KUKA KRL program: MyProgram_315().src

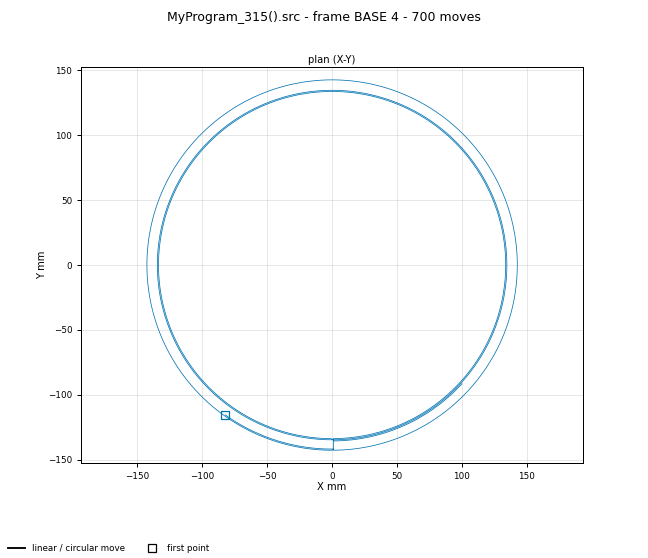
[picture p0: tool path of MyProgram_315().src in frame BASE 4, 700 of 700 moves have a stored position in this frame; points joined in program order, loops and branches not executed]
&ACCESS RVP
&REL 1
&PARAM TEMPLATE = C:\KRC\Roboter\Template\vorgabe
&PARAM EDITMASK = *
DEF MyProgram_315()
; ---- Setting reference (Base) ----
$BASE = BASE_DATA[4]

; --------------------------
; ---- Setting tool (TCP) ----
$TOOL = TOOL_DATA[3]
; --------------------------

$VEL.CP = VEL_APROX_PRINT
Startdeposition()
$VEL.CP = VEL_PRINT
LIN {X -82.35,Y -115.3687,Z 183,A -120.2522,B 3.9379,C 0.3327,E1 3.862,E2 213.1284} C_DIS
LIN {X -78.6424,Y -117.9272,Z 183,A -118.3809,B 3.9377,C 0.335,E1 3.8664,E2 211.2503} C_DIS
LIN {X -74.8735,Y -120.3553,Z 183,A -116.5285,B 3.9375,C 0.3372,E1 3.8708,E2 209.3924} C_DIS
LIN {X -70.8124,Y -122.7888,Z 183,A -114.6076,B 3.9373,C 0.3397,E1 3.8754,E2 207.4704} C_DIS
LIN {X -66.6703,Y -125.0867,Z 183,A -112.6373,B 3.9372,C 0.3416,E1 3.8802,E2 205.4924} C_DIS
LIN {X -63.0372,Y -126.954,Z 183,A -111.0289,B 3.937,C 0.3439,E1 3.8842,E2 203.8895} C_DIS
LIN {X -59.8265,Y -128.4982,Z 183,A -109.6089,B 3.9368,C 0.3456,E1 3.8878,E2 202.4722} C_DIS
LIN {X -56.4905,Y -129.9991,Z 183,A -108.1124,B 3.9367,C 0.3469,E1 3.8917,E2 200.973} C_DIS
LIN {X -53.5251,Y -131.2489,Z 183,A -106.7255,B 3.9367,C 0.3475,E1 3.8953,E2 199.5741} C_DIS
LIN {X -50.6002,Y -132.4053,Z 183,A -105.0533,B 3.9368,C 0.3452,E1 3.8998,E2 197.8465} C_DIS
LIN {X -46.7841,Y -133.7994,Z 183,A -103.1176,B 3.937,C 0.344,E1 3.905,E2 195.8696} C_DIS
LIN {X -41.3585,Y -135.5743,Z 183,A -101.5599,B 3.9362,C 0.3521,E1 3.9089,E2 194.4151} C_DIS
LIN {X -37.5342,Y -136.6841,Z 183,A -99.8325,B 3.9362,C 0.3521,E1 3.9136,E2 192.6712} C_DIS
LIN {X -34.185,Y -137.5602,Z 183,A -98.3691,B 3.9362,C 0.3523,E1 3.9176,E2 191.1985} C_DIS
LIN {X -30.1731,Y -138.494,Z 183,A -96.764,B 3.9362,C 0.3537,E1 3.9219,E2 189.6012} C_DIS
LIN {X -27.0139,Y -139.1451,Z 183,A -95.4028,B 3.9361,C 0.3537,E1 3.9257,E2 188.2317} C_DIS
LIN {X -23.267,Y -139.8199,Z 183,A -93.8958,B 3.9361,C 0.3545,E1 3.9298,E2 186.7286} C_DIS
LIN {X -18.7889,Y -140.4923,Z 183,A -92.1155,B 3.9359,C 0.3554,E1 3.9347,E2 184.9545} C_DIS
LIN {X -15.1936,Y -140.926,Z 183,A -90.5618,B 3.9359,C 0.3548,E1 3.9391,E2 183.3878} C_DIS
LIN {X -10.7309,Y -141.3366,Z 183,A -88.786,B 3.9359,C 0.3553,E1 3.944,E2 181.6162} C_DIS
LIN {X -6.3939,Y -141.6004,Z 183,A -86.9641,B 3.936,C 0.3547,E1 3.9491,E2 179.7846} C_DIS
LIN {X -2.1357,Y -141.7269,Z 183,A -85.3236,B 3.936,C 0.3554,E1 3.9537,E2 178.1545} C_DIS
LIN {X 0.9913,Y -141.7363,Z 183,A -84.3134,B 3.9357,C 0.3576,E1 3.9564,E2 177.1786} C_DIS
Enddeposition()
LIN {X 0.9913,Y -141.7363,Z 183,A -84.3134,B 3.9357,C 0.3576,E1 3.9564,E2 177.1786} C_DIS
Startdeposition()
$VEL.CP = VEL_PRINT
LIN {X 0.0025,Y -142.646,Z 183,A -85.0932,B 3.9352,C 0.3635,E1 3.954,E2 178.0429} C_DIS
LIN {X -3.4938,Y -142.6018,Z 183,A -86.4866,B 3.9352,C 0.3635,E1 3.9501,E2 179.4354} C_DIS
LIN {X -7.7044,Y -142.4366,Z 183,A -88.2171,B 3.9352,C 0.3639,E1 3.9453,E2 181.1718} C_DIS
LIN {X -11.5276,Y -142.178,Z 183,A -89.6214,B 3.9353,C 0.3626,E1 3.9414,E2 182.5582} C_DIS
LIN {X -15.0099,Y -141.852,Z 183,A -91.2226,B 3.9352,C 0.3642,E1 3.9369,E2 184.1869} C_DIS
LIN {X -19.1891,Y -141.3486,Z 183,A -92.7975,B 3.9352,C 0.3628,E1 3.9325,E2 185.7466} C_DIS
LIN {X -22.6498,Y -140.8363,Z 183,A -94.2297,B 3.9353,C 0.3626,E1 3.9286,E2 187.183} C_DIS
LIN {X -26.1124,Y -140.2348,Z 183,A -95.5706,B 3.9354,C 0.3615,E1 3.9249,E2 188.5147} C_DIS
LIN {X -28.8416,Y -139.698,Z 183,A -96.7574,B 3.9354,C 0.3616,E1 3.9216,E2 189.7113} C_DIS
LIN {X -32.9469,Y -138.7873,Z 183,A -98.6018,B 3.9354,C 0.3622,E1 3.9166,E2 191.5776} C_DIS
LIN {X -37.3426,Y -137.6701,Z 183,A -100.2942,B 3.9355,C 0.36,E1 3.912,E2 193.2527} C_DIS
LIN {X -40.2563,Y -136.8452,Z 183,A -101.5751,B 3.9355,C 0.3597,E1 3.9086,E2 194.5428} C_DIS
LIN {X -44.0427,Y -135.6755,Z 183,A -103.2725,B 3.9355,C 0.3595,E1 3.904,E2 196.2551} C_DIS
LIN {X -47.9851,Y -134.3307,Z 183,A -104.957,B 3.9357,C 0.3583,E1 3.8996,E2 197.9415} C_DIS
LIN {X -52.2995,Y -132.7114,Z 183,A -106.8391,B 3.9358,C 0.3569,E1 3.8946,E2 199.8282} C_DIS
LIN {X -56.8493,Y -130.8256,Z 183,A -108.7188,B 3.9361,C 0.3541,E1 3.8898,E2 201.6946} C_DIS
LIN {X -60.1958,Y -129.3202,Z 183,A -110.1929,B 3.9362,C 0.3526,E1 3.8861,E2 203.1689} C_DIS
LIN {X -63.3431,Y -127.8078,Z 183,A -111.6692,B 3.9362,C 0.3516,E1 3.8823,E2 204.6555} C_DIS
LIN {X -66.7705,Y -126.0518,Z 183,A -113.1503,B 3.9365,C 0.3493,E1 3.8787,E2 206.1278} C_DIS
LIN {X -70.1777,Y -124.1889,Z 183,A -114.8685,B 3.9365,C 0.3486,E1 3.8744,E2 207.8677} C_DIS
LIN {X -74.0833,Y -121.8994,Z 183,A -116.7206,B 3.9368,C 0.3464,E1 3.87,E2 209.7245} C_DIS
LIN {X -77.9926,Y -119.4361,Z 183,A -118.634,B 3.937,C 0.3442,E1 3.8655,E2 211.6458} C_DIS
LIN {X -81.8387,Y -116.8345,Z 183,A -120.4887,B 3.9372,C 0.3413,E1 3.8612,E2 213.499} C_DIS
LIN {X -85.3766,Y -114.2741,Z 183,A -122.2549,B 3.9374,C 0.3387,E1 3.8572,E2 215.2667} C_DIS
LIN {X -88.7267,Y -111.6928,Z 183,A -124.0258,B 3.9376,C 0.3364,E1 3.8533,E2 217.0474} C_DIS
LIN {X -92.1116,Y -108.9187,Z 183,A -125.838,B 3.9378,C 0.3338,E1 3.8494,E2 218.8669} C_DIS
LIN {X -95.4102,Y -106.041,Z 183,A -127.6362,B 3.9381,C 0.331,E1 3.8456,E2 220.6702} C_DIS
LIN {X -98.7395,Y -102.9478,Z 183,A -129.4764,B 3.9384,C 0.3277,E1 3.8419,E2 222.5122} C_DIS
LIN {X -101.9675,Y -99.7514,Z 183,A -131.3683,B 3.9386,C 0.3247,E1 3.8381,E2 224.4129} C_DIS
LIN {X -105.0998,Y -96.4454,Z 183,A -133.2356,B 3.9389,C 0.3213,E1 3.8346,E2 226.285} C_DIS
LIN {X -108.0049,Y -93.1807,Z 183,A -135.0551,B 3.9391,C 0.3181,E1 3.8312,E2 228.1127} C_DIS
LIN {X -111.047,Y -89.5335,Z 183,A -136.9938,B 3.9394,C 0.3143,E1 3.8278,E2 230.0551} C_DIS
LIN {X -113.7384,Y -86.0888,Z 183,A -138.7532,B 3.9397,C 0.3105,E1 3.8248,E2 231.8145} C_DIS
LIN {X -116.1196,Y -82.8489,Z 183,A -140.472,B 3.94,C 0.3076,E1 3.8219,E2 233.5468} C_DIS
LIN {X -118.6043,Y -79.2509,Z 183,A -142.2794,B 3.9403,C 0.304,E1 3.8191,E2 235.3604} C_DIS
LIN {X -120.9833,Y -75.5697,Z 183,A -144.079,B 3.9406,C 0.3001,E1 3.8164,E2 237.1648} C_DIS
LIN {X -123.2396,Y -71.8322,Z 183,A -145.927,B 3.9408,C 0.2965,E1 3.8137,E2 239.0248} C_DIS
LIN {X -125.38,Y -68.0268,Z 183,A -147.754,B 3.9411,C 0.2928,E1 3.8112,E2 240.8609} C_DIS
LIN {X -127.2528,Y -64.4509,Z 183,A -149.3448,B 3.9414,C 0.2885,E1 3.8092,E2 242.4468} C_DIS
LIN {X -128.9483,Y -60.9897,Z 183,A -150.9313,B 3.9417,C 0.2849,E1 3.8073,E2 244.0378} C_DIS
LIN {X -130.8258,Y -56.849,Z 183,A -152.914,B 3.9419,C 0.2812,E1 3.805,E2 246.0406} C_DIS
LIN {X -132.709,Y -52.3057,Z 183,A -154.9212,B 3.9423,C 0.2763,E1 3.8029,E2 248.0512} C_DIS
LIN {X -134.059,Y -48.7388,Z 183,A -156.5536,B 3.9425,C 0.2729,E1 3.8013,E2 249.6962} C_DIS
LIN {X -135.6246,Y -44.2019,Z 183,A -158.4657,B 3.9429,C 0.2677,E1 3.7996,E2 251.6052} C_DIS
LIN {X -136.7083,Y -40.7239,Z 183,A -159.9347,B 3.9431,C 0.2638,E1 3.7984,E2 253.0743} C_DIS
LIN {X -137.6658,Y -37.3588,Z 183,A -161.4756,B 3.9433,C 0.2608,E1 3.7973,E2 254.6323} C_DIS
LIN {X -138.7197,Y -33.2272,Z 183,A -163.1937,B 3.9436,C 0.2562,E1 3.7961,E2 256.3502} C_DIS
LIN {X -139.5524,Y -29.5406,Z 183,A -164.7326,B 3.9439,C 0.2521,E1 3.7952,E2 257.8909} C_DIS
LIN {X -140.2412,Y -26.079,Z 183,A -166.1968,B 3.9441,C 0.2485,E1 3.7944,E2 259.3605} C_DIS
LIN {X -140.8371,Y -22.6452,Z 183,A -167.6697,B 3.9444,C 0.2451,E1 3.7937,E2 260.8422} C_DIS
LIN {X -141.3475,Y -19.1975,Z 183,A -169.1215,B 3.9446,C 0.2415,E1 3.7931,E2 262.3001} C_DIS
LIN {X -141.7733,Y -15.7415,Z 183,A -170.5705,B 3.9448,C 0.2378,E1 3.7927,E2 263.7548} C_DIS
LIN {X -142.1148,Y -12.2755,Z 183,A -172.1312,B 3.945,C 0.2349,E1 3.7923,E2 265.3359} C_DIS
LIN {X -142.4358,Y -7.7214,Z 183,A -173.9354,B 3.9453,C 0.2295,E1 3.792,E2 267.135} C_DIS
LIN {X -142.5818,Y -4.2146,Z 183,A -175.3855,B 3.9455,C 0.2258,E1 3.7918,E2 268.5895} C_DIS
LIN {X -142.6476,Y -0.0075,Z 183,A -177.2034,B 3.9457,C 0.2218,E1 3.7918,E2 270.4232} C_DIS
LIN {X -142.6022,Y 3.4816,Z 183,A -178.6021,B 3.946,C 0.2178,E1 3.7918,E2 271.8204} C_DIS
LIN {X -142.441,Y 7.6183,Z 183,A 179.6198,B 3.9462,C 0.2138,E1 3.7921,E2 273.6124} C_DIS
LIN {X -142.1829,Y 11.4694,Z 183,A 178.1477,B 3.9464,C 0.2089,E1 3.7924,E2 275.0731} C_DIS
LIN {X -141.853,Y 15.0013,Z 183,A 176.5928,B 3.9466,C 0.2057,E1 3.7928,E2 276.644} C_DIS
LIN {X -141.3507,Y 19.1732,Z 183,A 174.8586,B 3.9468,C 0.2012,E1 3.7934,E2 278.3831} C_DIS
LIN {X -140.839,Y 22.6328,Z 183,A 173.4049,B 3.947,C 0.1976,E1 3.794,E2 279.8421} C_DIS
LIN {X -140.2388,Y 26.0914,Z 183,A 171.9887,B 3.9472,C 0.1937,E1 3.7947,E2 281.258} C_DIS
LIN {X -139.7058,Y 28.8029,Z 183,A 170.6646,B 3.9472,C 0.1919,E1 3.7955,E2 282.6092} C_DIS
LIN {X -138.7838,Y 32.9616,Z 183,A 168.8567,B 3.9475,C 0.1877,E1 3.7966,E2 284.4284} C_DIS
LIN {X -137.6667,Y 37.3555,Z 183,A 167.1157,B 3.9477,C 0.1823,E1 3.7978,E2 286.1576} C_DIS
LIN {X -136.7077,Y 40.7259,Z 183,A 165.6559,B 3.9479,C 0.1788,E1 3.799,E2 287.6231} C_DIS
LIN {X -135.6654,Y 44.0741,Z 183,A 164.0332,B 3.948,C 0.1762,E1 3.8004,E2 289.2725} C_DIS
LIN {X -134.3034,Y 48.061,Z 183,A 162.3117,B 3.9482,C 0.1719,E1 3.802,E2 290.9964} C_DIS
LIN {X -132.7108,Y 52.3011,Z 183,A 160.4077,B 3.9484,C 0.1676,E1 3.8039,E2 292.9099} C_DIS
LIN {X -130.8262,Y 56.848,Z 183,A 158.4915,B 3.9486,C 0.1621,E1 3.806,E2 294.8166} C_DIS
LIN {X -129.3279,Y 60.1791,Z 183,A 156.9927,B 3.9488,C 0.1585,E1 3.8077,E2 296.3183} C_DIS
LIN {X -127.8035,Y 63.3516,Z 183,A 155.477,B 3.9488,C 0.1556,E1 3.8096,E2 297.846} C_DIS
LIN {X -126.0351,Y 66.8022,Z 183,A 153.8636,B 3.949,C 0.152,E1 3.8117,E2 299.4654} C_DIS
LIN {X -123.933,Y 70.6278,Z 183,A 152.0311,B 3.9492,C 0.1482,E1 3.8142,E2 301.3067} C_DIS
LIN {X -121.6294,Y 74.525,Z 183,A 150.1752,B 3.9493,C 0.1441,E1 3.8169,E2 303.166} C_DIS
LIN {X -119.2914,Y 78.2133,Z 183,A 148.3566,B 3.9495,C 0.1403,E1 3.8196,E2 304.9915} C_DIS
LIN {X -116.8404,Y 81.8303,Z 183,A 146.541,B 3.9495,C 0.1367,E1 3.8225,E2 306.8134} C_DIS
LIN {X -114.2644,Y 85.3897,Z 183,A 144.7443,B 3.9497,C 0.1329,E1 3.8255,E2 308.6128} C_DIS
LIN {X -111.6942,Y 88.7248,Z 183,A 142.9703,B 3.9498,C 0.1297,E1 3.8285,E2 310.3959} C_DIS
LIN {X -108.9229,Y 92.1066,Z 183,A 141.1455,B 3.9499,C 0.1263,E1 3.8318,E2 312.2281} C_DIS
LIN {X -106.0397,Y 95.4115,Z 183,A 139.3422,B 3.95,C 0.1229,E1 3.8352,E2 314.0353} C_DIS
LIN {X -102.9541,Y 98.7329,Z 183,A 137.5179,B 3.9502,C 0.1193,E1 3.8387,E2 315.8587} C_DIS
LIN {X -99.8794,Y 101.8419,Z 183,A 135.7103,B 3.9502,C 0.1162,E1 3.8422,E2 317.6714} C_DIS
LIN {X -96.7026,Y 104.8634,Z 183,A 133.8965,B 3.9503,C 0.1132,E1 3.846,E2 319.4905} C_DIS
LIN {X -93.443,Y 107.7789,Z 183,A 132.023,B 3.9503,C 0.1108,E1 3.8499,E2 321.3775} C_DIS
LIN {X -89.8188,Y 110.8168,Z 183,A 130.146,B 3.9505,C 0.1073,E1 3.8539,E2 323.2502} C_DIS
LIN {X -86.3706,Y 113.525,Z 183,A 128.3193,B 3.9505,C 0.1048,E1 3.858,E2 325.0839} C_DIS
LIN {X -82.8502,Y 116.1186,Z 183,A 126.5424,B 3.9506,C 0.1021,E1 3.862,E2 326.8622} C_DIS
LIN {X -79.2527,Y 118.6031,Z 183,A 124.7541,B 3.9506,C 0.0996,E1 3.8662,E2 328.6532} C_DIS
LIN {X -75.5677,Y 120.9846,Z 183,A 122.9716,B 3.9508,C 0.0972,E1 3.8704,E2 330.437} C_DIS
LIN {X -71.8261,Y 123.2431,Z 183,A 121.146,B 3.9508,C 0.0953,E1 3.8748,E2 332.2703} C_DIS
LIN {X -68.0166,Y 125.3855,Z 183,A 119.3457,B 3.9508,C 0.0933,E1 3.8792,E2 334.075} C_DIS
LIN {X -64.4622,Y 127.247,Z 183,A 117.7885,B 3.9509,C 0.0909,E1 3.883,E2 335.624} C_DIS
LIN {X -60.9768,Y 128.9545,Z 183,A 116.2223,B 3.9509,C 0.0892,E1 3.887,E2 337.1902} C_DIS
LIN {X -56.8611,Y 130.8205,Z 183,A 114.2854,B 3.9509,C 0.0881,E1 3.892,E2 339.1413} C_DIS
LIN {X -52.3183,Y 132.7041,Z 183,A 112.3208,B 3.951,C 0.0861,E1 3.897,E2 341.1033} C_DIS
LIN {X -48.7543,Y 134.0534,Z 183,A 110.7188,B 3.951,C 0.0852,E1 3.9013,E2 342.7133} C_DIS
LIN {X -44.068,Y 135.6674,Z 183,A 108.8428,B 3.951,C 0.0827,E1 3.9062,E2 344.5735} C_DIS
LIN {X -40.7279,Y 136.7072,Z 183,A 107.4226,B 3.9511,C 0.0818,E1 3.91,E2 345.9948} C_DIS
LIN {X -37.3416,Y 137.6704,Z 183,A 105.9154,B 3.9511,C 0.0815,E1 3.9141,E2 347.513} C_DIS
LIN {X -33.6535,Y 138.617,Z 183,A 104.346,B 3.9511,C 0.0809,E1 3.9183,E2 349.0864} C_DIS
LIN {X -29.5672,Y 139.5466,Z 183,A 102.7687,B 3.9511,C 0.0792,E1 3.9226,E2 350.6495} C_DIS
LIN {X -26.1477,Y 140.2281,Z 183,A 101.3624,B 3.9511,C 0.0786,E1 3.9265,E2 352.0557} C_DIS
LIN {X -22.7049,Y 140.8272,Z 183,A 99.9472,B 3.9511,C 0.0781,E1 3.9304,E2 353.4717} C_DIS
LIN {X -19.1973,Y 141.3475,Z 183,A 98.501,B 3.9511,C 0.0779,E1 3.9344,E2 354.9199} C_DIS
LIN {X -15.7303,Y 141.7745,Z 183,A 97.096,B 3.9511,C 0.0775,E1 3.9383,E2 356.3244} C_DIS
LIN {X -12.2544,Y 142.1166,Z 183,A 95.5911,B 3.9511,C 0.0782,E1 3.9425,E2 357.8415} C_DIS
LIN {X -7.7279,Y 142.4355,Z 183,A 93.8546,B 3.9511,C 0.0773,E1 3.9473,E2 359.5662} C_DIS
LIN {X -4.2156,Y 142.5818,Z 183,A 92.3572,B 3.9511,C 0.078,E1 3.9515,E2 361.0738} C_DIS
LIN {X -0.0065,Y 142.646,Z 183,A 90.75,B 3.9511,C 0.0773,E1 3.956,E2 362.6697} C_DIS
LIN {X 3.4877,Y 142.602,Z 183,A 89.3573,B 3.9511,C 0.0774,E1 3.9599,E2 364.0604} C_DIS
LIN {X 7.1639,Y 142.4638,Z 183,A 87.7652,B 3.9511,C 0.0788,E1 3.9643,E2 365.6663} C_DIS
LIN {X 12.2339,Y 142.1184,Z 183,A 85.8331,B 3.9511,C 0.0784,E1 3.9697,E2 367.5839} C_DIS
LIN {X 16.7431,Y 141.6578,Z 183,A 83.9531,B 3.9511,C 0.0796,E1 3.9749,E2 369.4708} C_DIS
LIN {X 20.916,Y 141.1038,Z 183,A 82.394,B 3.9511,C 0.0792,E1 3.9792,E2 371.0127} C_DIS
LIN {X 24.3866,Y 140.5456,Z 183,A 80.9586,B 3.9511,C 0.0802,E1 3.9832,E2 372.4506} C_DIS
LIN {X 27.122,Y 140.0418,Z 183,A 79.8632,B 3.9511,C 0.0807,E1 3.9862,E2 373.5428} C_DIS
LIN {X 30.545,Y 139.3356,Z 183,A 78.3453,B 3.9511,C 0.0827,E1 3.9903,E2 375.0748} C_DIS
LIN {X 35.3323,Y 138.1986,Z 183,A 76.4792,B 3.9511,C 0.0831,E1 3.9954,E2 376.9264} C_DIS
LIN {X 39.0306,Y 137.2012,Z 183,A 74.9896,B 3.9511,C 0.0839,E1 3.9994,E2 378.4095} C_DIS
LIN {X 42.3592,Y 136.2104,Z 183,A 73.609,B 3.9511,C 0.085,E1 4.0031,E2 379.788} C_DIS
LIN {X 46.3155,Y 134.9155,Z 183,A 71.9558,B 3.9511,C 0.0865,E1 4.0074,E2 381.4384} C_DIS
LIN {X 50.3643,Y 133.4567,Z 183,A 70.2199,B 3.951,C 0.0883,E1 4.012,E2 383.1749} C_DIS
LIN {X 54.5937,Y 131.7832,Z 183,A 68.3183,B 3.9509,C 0.0912,E1 4.0169,E2 385.0858} C_DIS
LIN {X 58.6012,Y 130.0506,Z 183,A 66.7195,B 3.9509,C 0.0917,E1 4.021,E2 386.6645} C_DIS
LIN {X 61.7676,Y 128.5767,Z 183,A 65.3395,B 3.9509,C 0.0933,E1 4.0244,E2 388.0415} C_DIS
LIN {X 65.3625,Y 126.7887,Z 183,A 63.7084,B 3.9508,C 0.0956,E1 4.0285,E2 389.6749} C_DIS
LIN {X 68.7788,Y 124.9692,Z 183,A 62.1557,B 3.9508,C 0.0978,E1 4.0323,E2 391.2272} C_DIS
LIN {X 72.5889,Y 122.7953,Z 183,A 60.399,B 3.9507,C 0.1003,E1 4.0366,E2 392.9833} C_DIS
LIN {X 76.3148,Y 120.5146,Z 183,A 58.6918,B 3.9507,C 0.1026,E1 4.0406,E2 394.6844} C_DIS
LIN {X 79.9688,Y 118.1215,Z 183,A 56.986,B 3.9506,C 0.1049,E1 4.0446,E2 396.3839} C_DIS
LIN {X 83.8385,Y 115.4072,Z 183,A 55.1473,B 3.9505,C 0.1074,E1 4.0487,E2 398.215} C_DIS
LIN {X 87.4796,Y 112.6722,Z 183,A 53.3628,B 3.9505,C 0.1102,E1 4.0527,E2 399.9939} C_DIS
LIN {X 90.8907,Y 109.9389,Z 183,A 51.6353,B 3.9503,C 0.1131,E1 4.0564,E2 401.7179} C_DIS
LIN {X 94.1588,Y 107.154,Z 183,A 50.021,B 3.9503,C 0.1151,E1 4.0598,E2 403.3183} C_DIS
LIN {X 97.0585,Y 104.534,Z 183,A 48.3939,B 3.9502,C 0.1188,E1 4.0632,E2 404.953} C_DIS
LIN {X 100.2092,Y 101.5185,Z 183,A 46.6612,B 3.9501,C 0.1221,E1 4.0666,E2 406.6835} C_DIS
LIN {X 103.3076,Y 98.3631,Z 183,A 44.9537,B 3.95,C 0.125,E1 4.0699,E2 408.3824} C_DIS
LIN {X 106.2728,Y 95.1513,Z 183,A 43.2592,B 3.9499,C 0.1281,E1 4.0731,E2 410.0694} C_DIS
LIN {X 109.369,Y 91.5757,Z 183,A 41.4072,B 3.9498,C 0.1317,E1 4.0765,E2 411.9156} C_DIS
LIN {X 112.1152,Y 88.1923,Z 183,A 39.6991,B 3.9496,C 0.1351,E1 4.0794,E2 413.6187} C_DIS
LIN {X 114.8821,Y 84.5565,Z 183,A 37.9405,B 3.9496,C 0.1384,E1 4.0824,E2 415.3679} C_DIS
LIN {X 117.4262,Y 80.987,Z 183,A 36.2222,B 3.9494,C 0.1421,E1 4.0851,E2 417.0813} C_DIS
LIN {X 119.8522,Y 77.3516,Z 183,A 34.5204,B 3.9493,C 0.1456,E1 4.0877,E2 418.7768} C_DIS
LIN {X 122.082,Y 73.7812,Z 183,A 32.8734,B 3.9491,C 0.1492,E1 4.0901,E2 420.4186} C_DIS
LIN {X 124.3638,Y 69.8666,Z 183,A 31.1316,B 3.949,C 0.1528,E1 4.0925,E2 422.151} C_DIS
LIN {X 126.3848,Y 66.1364,Z 183,A 29.5107,B 3.9489,C 0.1561,E1 4.0946,E2 423.7616} C_DIS
LIN {X 128.1961,Y 62.5559,Z 183,A 27.9669,B 3.9487,C 0.1594,E1 4.0965,E2 425.2972} C_DIS
LIN {X 129.8393,Y 59.0732,Z 183,A 26.31,B 3.9485,C 0.1647,E1 4.0985,E2 426.9692} C_DIS
LIN {X 131.5102,Y 55.2474,Z 183,A 24.7343,B 3.9484,C 0.1678,E1 4.1002,E2 428.5324} C_DIS
LIN {X 133.2658,Y 50.8735,Z 183,A 22.8846,B 3.9482,C 0.1723,E1 4.1021,E2 430.3774} C_DIS
LIN {X 134.6065,Y 47.2069,Z 183,A 21.3487,B 3.948,C 0.1761,E1 4.1035,E2 431.9099} C_DIS
LIN {X 135.9833,Y 43.079,Z 183,A 19.8149,B 3.948,C 0.1782,E1 4.1048,E2 433.4165} C_DIS
LIN {X 137.0065,Y 39.7055,Z 183,A 18.4481,B 3.9478,C 0.1815,E1 4.1059,E2 434.7776} C_DIS
LIN {X 138.0656,Y 35.8563,Z 183,A 16.7654,B 3.9475,C 0.1868,E1 4.1071,E2 436.4716} C_DIS
LIN {X 139.1746,Y 31.2708,Z 183,A 15.0712,B 3.9475,C 0.1896,E1 4.1082,E2 438.1404} C_DIS
LIN {X 139.898,Y 27.8587,Z 183,A 13.7201,B 3.9472,C 0.1929,E1 4.109,E2 439.4857} C_DIS
LIN {X 140.5388,Y 24.4246,Z 183,A 12.3663,B 3.9471,C 0.1962,E1 4.1096,E2 440.8339} C_DIS
LIN {X 141.2482,Y 19.9058,Z 183,A 10.5555,B 3.9468,C 0.201,E1 4.1104,E2 442.6423} C_DIS
LIN {X 141.7743,Y 15.732,Z 183,A 8.9443,B 3.9466,C 0.2048,E1 4.1109,E2 444.2442} C_DIS
LIN {X 142.1178,Y 12.2398,Z 183,A 7.4912,B 3.9464,C 0.2093,E1 4.1113,E2 445.704} C_DIS
LIN {X 142.4363,Y 7.7104,Z 183,A 5.8187,B 3.9462,C 0.2126,E1 4.1116,E2 447.3577} C_DIS
LIN {X 142.6016,Y 3.5031,Z 183,A 4.1212,B 3.946,C 0.2175,E1 4.1117,E2 449.0571} C_DIS
LIN {X 142.6426,Y -0.7871,Z 183,A 2.4653,B 3.9457,C 0.2215,E1 4.1117,E2 450.7052} C_DIS
LIN {X 142.5473,Y -5.2571,Z 183,A 0.6958,B 3.9455,C 0.2263,E1 4.1117,E2 452.4725} C_DIS
LIN {X 142.3093,Y -9.7809,Z 183,A -0.9673,B 3.9453,C 0.2295,E1 4.1113,E2 454.116} C_DIS
LIN {X 142.0566,Y -12.9471,Z 183,A -2.2735,B 3.9451,C 0.2335,E1 4.111,E2 455.4273} C_DIS
LIN {X 141.6577,Y -16.7439,Z 183,A -3.759,B 3.9448,C 0.2372,E1 4.1106,E2 456.9074} C_DIS
LIN {X 141.1008,Y -20.9369,Z 183,A -5.2976,B 3.9447,C 0.24,E1 4.11,E2 458.426} C_DIS
LIN {X 140.3703,Y -25.3663,Z 183,A -7.0475,B 3.9444,C 0.2444,E1 4.1091,E2 460.1701} C_DIS
LIN {X 139.699,Y -28.8363,Z 183,A -8.4144,B 3.9442,C 0.2477,E1 4.1084,E2 461.5311} C_DIS
LIN {X 138.7855,Y -32.9545,Z 183,A -10.1869,B 3.9438,C 0.2534,E1 4.1073,E2 463.3153} C_DIS
LIN {X 137.6699,Y -37.3437,Z 183,A -11.8046,B 3.9437,C 0.2559,E1 4.1062,E2 464.9074} C_DIS
LIN {X 136.7119,Y -40.7117,Z 183,A -13.1686,B 3.9435,C 0.2592,E1 4.1051,E2 466.2669} C_DIS
LIN {X 135.6774,Y -44.0368,Z 183,A -14.6582,B 3.9431,C 0.2641,E1 4.1038,E2 467.7698} C_DIS
LIN {X 134.3301,Y -47.9868,Z 183,A -16.2733,B 3.9429,C 0.2679,E1 4.1023,E2 469.378} C_DIS
LIN {X 132.7106,Y -52.3016,Z 183,A -18.0733,B 3.9426,C 0.2722,E1 4.1005,E2 471.1727} C_DIS
LIN {X 130.8247,Y -56.8514,Z 183,A -19.8673,B 3.9424,C 0.2752,E1 4.0986,E2 472.9433} C_DIS
LIN {X 129.3138,Y -60.2097,Z 183,A -21.2811,B 3.9422,C 0.2782,E1 4.097,E2 474.3496} C_DIS
LIN {X 127.805,Y -63.3486,Z 183,A -22.6856,B 3.9419,C 0.2819,E1 4.0953,E2 475.756} C_DIS
LIN {X 126.0536,Y -66.7671,Z 183,A -24.1788,B 3.9417,C 0.2852,E1 4.0933,E2 477.2438} C_DIS
LIN {X 123.9527,Y -70.5934,Z 183,A -25.9055,B 3.9414,C 0.2893,E1 4.091,E2 478.9684} C_DIS
LIN {X 121.6287,Y -74.5262,Z 183,A -27.6627,B 3.9411,C 0.2929,E1 4.0885,E2 480.7167} C_DIS
LIN {X 119.2881,Y -78.2182,Z 183,A -29.3744,B 3.9408,C 0.2966,E1 4.0859,E2 482.4239} C_DIS
LIN {X 116.8354,Y -81.8375,Z 183,A -31.135,B 3.9405,C 0.3009,E1 4.0831,E2 484.1865} C_DIS
LIN {X 114.0501,Y -85.6759,Z 183,A -32.9572,B 3.9402,C 0.3043,E1 4.0801,E2 485.9991} C_DIS
LIN {X 111.3707,Y -89.1314,Z 183,A -34.6674,B 3.94,C 0.3078,E1 4.0771,E2 487.7045} C_DIS
LIN {X 108.5656,Y -92.5269,Z 183,A -36.3236,B 3.9398,C 0.3104,E1 4.0742,E2 489.3469} C_DIS
LIN {X 105.7297,Y -95.7545,Z 183,A -38.0262,B 3.9395,C 0.3139,E1 4.071,E2 491.0477} C_DIS
LIN {X 102.7689,Y -98.9263,Z 183,A -39.737,B 3.9392,C 0.3172,E1 4.0678,E2 492.7556} C_DIS
LIN {X 99.6151,Y -102.1011,Z 183,A -41.4796,B 3.939,C 0.3203,E1 4.0643,E2 494.4921} C_DIS
LIN {X 96.4524,Y -105.0935,Z 183,A -43.198,B 3.9387,C 0.3235,E1 4.0608,E2 496.2079} C_DIS
LIN {X 93.1977,Y -107.9902,Z 183,A -44.8898,B 3.9385,C 0.3262,E1 4.0573,E2 497.8931} C_DIS
LIN {X 89.8077,Y -110.8258,Z 183,A -46.6298,B 3.9382,C 0.3292,E1 4.0535,E2 499.6298} C_DIS
LIN {X 86.3849,Y -113.5141,Z 183,A -48.3649,B 3.938,C 0.3322,E1 4.0497,E2 501.3644} C_DIS
LIN {X 82.8797,Y -116.0976,Z 183,A -50.06,B 3.9378,C 0.3347,E1 4.0459,E2 503.0536} C_DIS
LIN {X 79.2906,Y -118.5778,Z 183,A -51.7816,B 3.9376,C 0.3373,E1 4.0419,E2 504.7724} C_DIS
LIN {X 75.4673,Y -121.047,Z 183,A -53.5372,B 3.9374,C 0.3394,E1 4.0378,E2 506.5194} C_DIS
LIN {X 71.6256,Y -123.3592,Z 183,A -55.3232,B 3.9371,C 0.342,E1 4.0335,E2 508.3047} C_DIS
LIN {X 67.7118,Y -125.5502,Z 183,A -57.0831,B 3.9369,C 0.3442,E1 4.0292,E2 510.0603} C_DIS
LIN {X 64.4574,Y -127.2495,Z 183,A -58.5108,B 3.9369,C 0.3458,E1 4.0257,E2 511.4825} C_DIS
LIN {X 60.9784,Y -128.9537,Z 183,A -60.0036,B 3.9367,C 0.3472,E1 4.0219,E2 512.9678} C_DIS
LIN {X 58.1268,Y -130.2628,Z 183,A -61.2856,B 3.9365,C 0.3491,E1 4.0186,E2 514.2536} C_DIS
LIN {X 54.5907,Y -131.7845,Z 183,A -62.8657,B 3.9363,C 0.3513,E1 4.0146,E2 515.8396} C_DIS
LIN {X 50.3777,Y -133.4517,Z 183,A -64.5539,B 3.9363,C 0.352,E1 4.0102,E2 517.5109} C_DIS
LIN {X 46.4236,Y -134.878,Z 183,A -66.2207,B 3.9361,C 0.3536,E1 4.0058,E2 519.1758} C_DIS
LIN {X 43.0796,Y -135.9831,Z 183,A -67.6169,B 3.9361,C 0.3548,E1 4.0021,E2 520.5705} C_DIS
LIN {X 39.7056,Y -137.0065,Z 183,A -69.1236,B 3.9358,C 0.3571,E1 3.998,E2 522.0906} C_DIS
LIN {X 35.3426,Y -138.196,Z 183,A -70.8149,B 3.9358,C 0.3573,E1 3.9935,E2 523.7658} C_DIS
LIN {X 31.3774,Y -139.1503,Z 183,A -72.4419,B 3.9357,C 0.3585,E1 3.9891,E2 525.3923} C_DIS
LIN {X 27.837,Y -139.9024,Z 183,A -73.8687,B 3.9357,C 0.3593,E1 3.9852,E2 526.8162} C_DIS
LIN {X 24.4026,Y -140.5427,Z 183,A -75.2571,B 3.9355,C 0.36,E1 3.9814,E2 528.2034} C_DIS
LIN {X 19.9259,Y -141.2453,Z 183,A -77.1052,B 3.9355,C 0.3613,E1 3.9763,E2 530.0564} C_DIS
LIN {X 15.7235,Y -141.7752,Z 183,A -78.775,B 3.9354,C 0.3618,E1 3.9716,E2 531.7228} C_DIS
LIN {X 12.2454,Y -142.1174,Z 183,A -80.2673,B 3.9352,C 0.3632,E1 3.9674,E2 533.228} C_DIS
LIN {X 7.7215,Y -142.4358,Z 183,A -81.9908,B 3.9352,C 0.3629,E1 3.9627,E2 534.939} C_DIS
LIN {X 4.2511,Y -142.5808,Z 183,A -83.479,B 3.9352,C 0.3641,E1 3.9585,E2 536.4407} C_DIS
LIN {X 0.9972,Y -142.6395,Z 183,A -84.3846,B 3.9355,C 0.3605,E1 3.9561,E2 537.2915} C_DIS
Enddeposition()
LIN {X 0.9679,Y -133.7011,Z 184,A -84.8201,B 3.7652,C 0.3379,E1 3.7837,E2 537.5155} C_DIS
Startdeposition()
$VEL.CP = VEL_PRINT
LIN {X 4.9139,Y -133.6145,Z 184,A -82.3604,B 3.7659,C 0.3309,E1 3.7909,E2 534.9564} C_DIS
LIN {X 9.0962,Y -133.3962,Z 184,A -80.5448,B 3.7659,C 0.3302,E1 3.796,E2 533.1373} C_DIS
LIN {X 13.0754,Y -133.0639,Z 184,A -79.0141,B 3.7659,C 0.3311,E1 3.8002,E2 531.6289} C_DIS
LIN {X 16.365,Y -132.7001,Z 184,A -77.6114,B 3.7659,C 0.3305,E1 3.804,E2 530.2274} C_DIS
LIN {X 19.6102,Y -132.2603,Z 184,A -76.2198,B 3.7659,C 0.3299,E1 3.8079,E2 528.8366} C_DIS
LIN {X 22.8429,Y -131.7405,Z 184,A -74.8055,B 3.766,C 0.3289,E1 3.8118,E2 527.42} C_DIS
LIN {X 26.0646,Y -131.1405,Z 184,A -73.4095,B 3.7661,C 0.328,E1 3.8156,E2 526.0242} C_DIS
LIN {X 29.9874,Y -130.2982,Z 184,A -71.7232,B 3.7662,C 0.3271,E1 3.8202,E2 524.3411} C_DIS
LIN {X 33.1715,Y -129.5243,Z 184,A -70.3342,B 3.7662,C 0.326,E1 3.824,E2 522.9532} C_DIS
LIN {X 36.3354,Y -128.6726,Z 184,A -68.9465,B 3.7664,C 0.3249,E1 3.8277,E2 521.5667} C_DIS
LIN {X 39.683,Y -127.6808,Z 184,A -67.4705,B 3.7664,C 0.3237,E1 3.8317,E2 520.0923} C_DIS
LIN {X 43.0012,Y -126.603,Z 184,A -65.8461,B 3.7667,C 0.3209,E1 3.836,E2 518.4503} C_DIS
LIN {X 46.5935,Y -125.3233,Z 184,A -64.3844,B 3.7667,C 0.3209,E1 3.8398,E2 517.0096} C_DIS
LIN {X 50.3106,Y -123.8779,Z 184,A -62.6982,B 3.7669,C 0.319,E1 3.8442,E2 515.3252} C_DIS
LIN {X 53.5297,Y -122.5218,Z 184,A -61.0933,B 3.7671,C 0.3161,E1 3.8483,E2 513.7053} C_DIS
LIN {X 57.1603,Y -120.8707,Z 184,A -59.5538,B 3.7671,C 0.3155,E1 3.8522,E2 512.1865} C_DIS
LIN {X 60.1047,Y -119.4343,Z 184,A -58.1778,B 3.7673,C 0.3139,E1 3.8556,E2 510.813} C_DIS
LIN {X 63.1179,Y -117.8705,Z 184,A -56.7615,B 3.7675,C 0.3122,E1 3.8591,E2 509.4006} C_DIS
LIN {X 66.4973,Y -115.9977,Z 184,A -55.1187,B 3.7677,C 0.3098,E1 3.8631,E2 507.7582} C_DIS
LIN {X 69.4683,Y -114.2434,Z 184,A -53.5345,B 3.7679,C 0.3064,E1 3.8669,E2 506.1593} C_DIS
LIN {X 72.8121,Y -112.1413,Z 184,A -51.9684,B 3.768,C 0.305,E1 3.8706,E2 504.6082} C_DIS
LIN {X 76.2275,Y -109.8484,Z 184,A -50.2902,B 3.7682,C 0.3029,E1 3.8744,E2 502.9395} C_DIS
LIN {X 78.9118,Y -107.9366,Z 184,A -48.9198,B 3.7684,C 0.3008,E1 3.8775,E2 501.5733} C_DIS
LIN {X 81.8933,Y -105.6919,Z 184,A -47.2769,B 3.7686,C 0.2975,E1 3.8812,E2 499.9235} C_DIS
LIN {X 85.1711,Y -103.0688,Z 184,A -45.4762,B 3.7689,C 0.2941,E1 3.8851,E2 498.1212} C_DIS
LIN {X 88.5676,Y -100.1652,Z 184,A -43.6556,B 3.7691,C 0.2914,E1 3.8889,E2 496.3111} C_DIS
LIN {X 91.8598,Y -97.1549,Z 184,A -41.7924,B 3.7694,C 0.288,E1 3.8927,E2 494.4526} C_DIS
LIN {X 94.8634,Y -94.2243,Z 184,A -40.0611,B 3.7696,C 0.285,E1 3.8961,E2 492.7284} C_DIS
LIN {X 97.6433,Y -91.3409,Z 184,A -38.3187,B 3.7699,C 0.2811,E1 3.8995,E2 490.9813} C_DIS
LIN {X 100.7078,Y -87.9501,Z 184,A -36.4859,B 3.7701,C 0.2782,E1 3.9029,E2 489.1629} C_DIS
LIN {X 103.353,Y -84.8264,Z 184,A -34.7533,B 3.7704,C 0.2745,E1 3.906,E2 487.4316} C_DIS
LIN {X 105.9006,Y -81.624,Z 184,A -33.1221,B 3.7706,C 0.2718,E1 3.9088,E2 485.8146} C_DIS
LIN {X 108.3816,Y -78.2991,Z 184,A -31.4169,B 3.7708,C 0.2685,E1 3.9116,E2 484.1172} C_DIS
LIN {X 110.2633,Y -75.626,Z 184,A -29.9338,B 3.7711,C 0.2642,E1 3.9139,E2 482.6223} C_DIS
LIN {X 112.4678,Y -72.3073,Z 184,A -28.3358,B 3.7713,C 0.2613,E1 3.9164,E2 481.0369} C_DIS
LIN {X 114.6816,Y -68.7425,Z 184,A -26.5535,B 3.7716,C 0.257,E1 3.919,E2 479.2551} C_DIS
LIN {X 116.6747,Y -65.302,Z 184,A -25.0168,B 3.7718,C 0.2546,E1 3.921,E2 477.7383} C_DIS
LIN {X 118.2368,Y -62.4251,Z 184,A -23.6671,B 3.772,C 0.2517,E1 3.9228,E2 476.394} C_DIS
LIN {X 119.7466,Y -59.4779,Z 184,A -22.241,B 3.7722,C 0.248,E1 3.9246,E2 474.9659} C_DIS
LIN {X 121.2601,Y -56.3275,Z 184,A -20.9069,B 3.7724,C 0.2459,E1 3.9262,E2 473.6513} C_DIS
LIN {X 122.5188,Y -53.5365,Z 184,A -19.5207,B 3.7726,C 0.2417,E1 3.9278,E2 472.2547} C_DIS
LIN {X 124.149,Y -49.6379,Z 184,A -17.7164,B 3.7729,C 0.2369,E1 3.9297,E2 470.4497} C_DIS
LIN {X 125.5671,Y -45.9355,Z 184,A -16.1928,B 3.7731,C 0.2344,E1 3.9311,E2 468.9469} C_DIS
LIN {X 126.7154,Y -42.6636,Z 184,A -14.6118,B 3.7734,C 0.2293,E1 3.9326,E2 467.3527} C_DIS
LIN {X 127.9478,Y -38.8106,Z 184,A -13.0814,B 3.7736,C 0.2269,E1 3.9338,E2 465.8465} C_DIS
LIN {X 128.8612,Y -35.6613,Z 184,A -11.7272,B 3.7737,C 0.2236,E1 3.9349,E2 464.4976} C_DIS
LIN {X 129.7158,Y -32.417,Z 184,A -10.3478,B 3.7739,C 0.2203,E1 3.9358,E2 463.1245} C_DIS
LIN {X 130.6123,Y -28.5903,Z 184,A -8.7116,B 3.7742,C 0.2162,E1 3.9368,E2 461.493} C_DIS
LIN {X 131.314,Y -25.1686,Z 184,A -7.2719,B 3.7744,C 0.2127,E1 3.9376,E2 460.0594} C_DIS
LIN {X 131.8913,Y -21.9434,Z 184,A -5.9594,B 3.7745,C 0.2098,E1 3.9382,E2 458.7573} C_DIS
LIN {X 132.3589,Y -18.9202,Z 184,A -4.6569,B 3.7747,C 0.2062,E1 3.9388,E2 457.4549} C_DIS
LIN {X 132.8085,Y -15.4569,Z 184,A -3.0767,B 3.775,C 0.201,E1 3.9393,E2 455.8631} C_DIS
LIN {X 133.2119,Y -11.4672,Z 184,A -1.4539,B 3.7752,C 0.1973,E1 3.9397,E2 454.251} C_DIS
LIN {X 133.4963,Y -7.4935,Z 184,A 0.2881,B 3.7755,C 0.192,E1 3.94,E2 452.5035} C_DIS
LIN {X 133.68,Y -2.588,Z 184,A 2.1704,B 3.7757,C 0.1886,E1 3.9402,E2 450.6474} C_DIS
LIN {X 133.7027,Y 0.6833,Z 184,A 3.496,B 3.7758,C 0.1855,E1 3.9402,E2 449.3303} C_DIS
LIN {X 133.6142,Y 4.9214,Z 184,A 5.3501,B 3.7761,C 0.1799,E1 3.94,E2 447.4703} C_DIS
LIN {X 133.3951,Y 9.1117,Z 184,A 7.1068,B 3.7763,C 0.1753,E1 3.9397,E2 445.7177} C_DIS
LIN {X 133.0611,Y 13.1039,Z 184,A 8.7303,B 3.7765,C 0.1716,E1 3.9393,E2 444.1047} C_DIS
LIN {X 132.5814,Y 17.2924,Z 184,A 10.3428,B 3.7765,C 0.1687,E1 3.9387,E2 442.5151} C_DIS
LIN {X 132.118,Y 20.5351,Z 184,A 11.6768,B 3.7767,C 0.1655,E1 3.9382,E2 441.1889} C_DIS
LIN {X 131.6136,Y 23.5517,Z 184,A 12.9577,B 3.7769,C 0.1622,E1 3.9376,E2 439.9109} C_DIS
LIN {X 130.9541,Y 26.9806,Z 184,A 14.5247,B 3.7771,C 0.1573,E1 3.9367,E2 438.3343} C_DIS
LIN {X 129.9198,Y 31.5867,Z 184,A 16.3494,B 3.7772,C 0.1539,E1 3.9356,E2 436.533} C_DIS
LIN {X 129.1061,Y 34.7638,Z 184,A 17.7051,B 3.7774,C 0.1506,E1 3.9346,E2 435.1826} C_DIS
LIN {X 128.2158,Y 37.916,Z 184,A 19.1829,B 3.7775,C 0.146,E1 3.9335,E2 433.6949} C_DIS
LIN {X 126.9556,Y 41.9423,Z 184,A 20.8093,B 3.7776,C 0.1431,E1 3.9321,E2 432.09} C_DIS
LIN {X 125.8844,Y 45.0554,Z 184,A 22.1663,B 3.7778,C 0.1399,E1 3.9308,E2 430.7388} C_DIS
LIN {X 124.7428,Y 48.1261,Z 184,A 23.6529,B 3.7779,C 0.1353,E1 3.9293,E2 429.2414} C_DIS
LIN {X 123.2522,Y 51.8243,Z 184,A 25.1975,B 3.778,C 0.1326,E1 3.9277,E2 427.7163} C_DIS
LIN {X 121.5627,Y 55.6732,Z 184,A 26.909,B 3.7782,C 0.129,E1 3.9258,E2 426.015} C_DIS
LIN {X 120.1629,Y 58.6341,Z 184,A 28.2634,B 3.7782,C 0.1259,E1 3.9242,E2 424.666} C_DIS
LIN {X 118.6807,Y 61.5797,Z 184,A 29.614,B 3.7784,C 0.123,E1 3.9224,E2 423.3225} C_DIS
LIN {X 117.1355,Y 64.4723,Z 184,A 31.1308,B 3.7785,C 0.1183,E1 3.9204,E2 421.7915} C_DIS
LIN {X 115.1536,Y 67.9485,Z 184,A 32.6858,B 3.7785,C 0.1158,E1 3.9182,E2 420.2554} C_DIS
LIN {X 112.9626,Y 71.5317,Z 184,A 34.4015,B 3.7787,C 0.1123,E1 3.9157,E2 418.5494} C_DIS
LIN {X 111.1764,Y 74.2772,Z 184,A 35.7588,B 3.7787,C 0.1095,E1 3.9137,E2 417.1972} C_DIS
LIN {X 108.9172,Y 77.5525,Z 184,A 37.4856,B 3.7789,C 0.1053,E1 3.9109,E2 415.4673} C_DIS
LIN {X 106.4081,Y 80.9612,Z 184,A 39.2492,B 3.7789,C 0.1016,E1 3.9079,E2 413.7093} C_DIS
LIN {X 103.8709,Y 84.1915,Z 184,A 40.9726,B 3.7791,C 0.0981,E1 3.9049,E2 411.99} C_DIS
LIN {X 101.0111,Y 87.6026,Z 184,A 42.8334,B 3.7791,C 0.0944,E1 3.9016,E2 410.1344} C_DIS
LIN {X 98.2068,Y 90.7349,Z 184,A 44.5544,B 3.7793,C 0.0914,E1 3.8984,E2 408.4227} C_DIS
LIN {X 95.4444,Y 93.6357,Z 184,A 46.2261,B 3.7793,C 0.0883,E1 3.8951,E2 406.7561} C_DIS
LIN {X 92.4591,Y 96.5847,Z 184,A 47.9691,B 3.7793,C 0.0853,E1 3.8916,E2 405.0196} C_DIS
LIN {X 89.4437,Y 99.3842,Z 184,A 49.6979,B 3.7795,C 0.0822,E1 3.8881,E2 403.2946} C_DIS
LIN {X 86.4402,Y 102.0069,Z 184,A 51.3721,B 3.7795,C 0.0793,E1 3.8845,E2 401.6244} C_DIS
LIN {X 83.1898,Y 104.6745,Z 184,A 53.1018,B 3.7795,C 0.0767,E1 3.8808,E2 399.9033} C_DIS
LIN {X 80.2328,Y 106.9585,Z 184,A 54.7568,B 3.7796,C 0.0734,E1 3.8771,E2 398.2418} C_DIS
LIN {X 76.9806,Y 109.3219,Z 184,A 56.2963,B 3.7796,C 0.0723,E1 3.8737,E2 396.7241} C_DIS
LIN {X 73.6858,Y 111.5694,Z 184,A 57.9633,B 3.7797,C 0.0699,E1 3.8698,E2 395.0622} C_DIS
LIN {X 70.4636,Y 113.6319,Z 184,A 59.6372,B 3.7797,C 0.067,E1 3.8658,E2 393.3842} C_DIS
LIN {X 67.3332,Y 115.5149,Z 184,A 61.2475,B 3.7798,C 0.0642,E1 3.862,E2 391.7686} C_DIS
LIN {X 63.88,Y 117.4592,Z 184,A 62.8259,B 3.7798,C 0.0629,E1 3.8581,E2 390.2047} C_DIS
LIN {X 60.9461,Y 119.006,Z 184,A 64.1653,B 3.7798,C 0.0617,E1 3.8548,E2 388.875} C_DIS
LIN {X 57.7508,Y 120.5886,Z 184,A 65.7743,B 3.7798,C 0.059,E1 3.8508,E2 387.2565} C_DIS
LIN {X 53.5318,Y 122.5209,Z 184,A 67.6825,B 3.7799,C 0.0573,E1 3.8459,E2 385.3582} C_DIS
LIN {X 49.6515,Y 124.1436,Z 184,A 69.5143,B 3.7799,C 0.0549,E1 3.8412,E2 383.5232} C_DIS
LIN {X 45.9332,Y 125.5679,Z 184,A 71.0809,B 3.7799,C 0.0544,E1 3.8371,E2 381.9735} C_DIS
LIN {X 42.1307,Y 126.8928,Z 184,A 72.8122,B 3.7799,C 0.0526,E1 3.8325,E2 380.2419} C_DIS
LIN {X 38.8478,Y 127.9364,Z 184,A 74.2399,B 3.78,C 0.0517,E1 3.8287,E2 378.8203} C_DIS
LIN {X 35.0998,Y 129.0165,Z 184,A 75.9962,B 3.78,C 0.0496,E1 3.824,E2 377.0543} C_DIS
LIN {X 30.897,Y 130.0861,Z 184,A 77.8735,B 3.78,C 0.048,E1 3.8189,E2 375.1752} C_DIS
LIN {X 27.0042,Y 130.9493,Z 184,A 79.485,B 3.78,C 0.0477,E1 3.8145,E2 373.5757} C_DIS
LIN {X 23.5566,Y 131.6127,Z 184,A 80.9203,B 3.78,C 0.0473,E1 3.8106,E2 372.1491} C_DIS
LIN {X 20.5403,Y 132.1172,Z 184,A 82.2231,B 3.78,C 0.0467,E1 3.807,E2 370.8477} C_DIS
LIN {X 17.2967,Y 132.5808,Z 184,A 83.6438,B 3.78,C 0.0459,E1 3.8031,E2 369.4255} C_DIS
LIN {X 13.1166,Y 133.0599,Z 184,A 85.4226,B 3.78,C 0.0454,E1 3.7981,E2 367.6502} C_DIS
LIN {X 9.1255,Y 133.3941,Z 184,A 87.1012,B 3.78,C 0.0452,E1 3.7935,E2 365.9768} C_DIS
LIN {X 4.928,Y 133.6139,Z 184,A 89.046,B 3.7801,C 0.0436,E1 3.788,E2 364.0155} C_DIS
LIN {X 0.732,Y 133.7026,Z 184,A 90.6701,B 3.7801,C 0.0448,E1 3.7835,E2 362.4129} C_DIS
LIN {X -2.5396,Y 133.6808,Z 184,A 92.1033,B 3.7801,C 0.0445,E1 3.7795,E2 360.9767} C_DIS
LIN {X -5.63,Y 133.5866,Z 184,A 93.4416,B 3.7801,C 0.0445,E1 3.7758,E2 359.6374} C_DIS
LIN {X -9.1142,Y 133.3949,Z 184,A 95.1009,B 3.7801,C 0.0433,E1 3.7711,E2 357.9594} C_DIS
LIN {X -13.0906,Y 133.0624,Z 184,A 96.7781,B 3.7801,C 0.0438,E1 3.7664,E2 356.2869} C_DIS
LIN {X -17.2897,Y 132.5818,Z 184,A 98.4683,B 3.7801,C 0.0452,E1 3.7618,E2 354.6119} C_DIS
LIN {X -20.5331,Y 132.1183,Z 184,A 99.8357,B 3.7801,C 0.0459,E1 3.758,E2 353.2496} C_DIS
LIN {X -23.5503,Y 131.6139,Z 184,A 101.2405,B 3.7801,C 0.0457,E1 3.7541,E2 351.8343} C_DIS
LIN {X -27.6787,Y 130.8091,Z 184,A 103.1707,B 3.7801,C 0.0457,E1 3.7488,E2 349.89} C_DIS
LIN {X -31.5854,Y 129.9201,Z 184,A 104.7375,B 3.7801,C 0.0477,E1 3.7446,E2 348.3419} C_DIS
LIN {X -34.7607,Y 129.1069,Z 184,A 106.1551,B 3.7801,C 0.0485,E1 3.7407,E2 346.9236} C_DIS
LIN {X -37.915,Y 128.2161,Z 184,A 107.5991,B 3.7801,C 0.0492,E1 3.7369,E2 345.4758} C_DIS
LIN {X -41.9486,Y 126.9535,Z 184,A 109.4033,B 3.7801,C 0.0507,E1 3.7321,E2 343.6735} C_DIS
LIN {X -45.0365,Y 125.8912,Z 184,A 110.8183,B 3.7801,C 0.0518,E1 3.7283,E2 342.2575} C_DIS
LIN {X -48.0954,Y 124.7547,Z 184,A 112.374,B 3.78,C 0.052,E1 3.7242,E2 340.6841} C_DIS
LIN {X -51.7481,Y 123.284,Z 184,A 113.9733,B 3.78,C 0.0543,E1 3.7201,E2 339.0963} C_DIS
LIN {X -55.5944,Y 121.5991,Z 184,A 115.7984,B 3.78,C 0.0561,E1 3.7155,E2 337.2694} C_DIS
LIN {X -58.6415,Y 120.1592,Z 184,A 117.2344,B 3.78,C 0.0578,E1 3.7118,E2 335.8353} C_DIS
LIN {X -62.009,Y 118.4552,Z 184,A 118.6909,B 3.7799,C 0.0608,E1 3.7083,E2 334.399} C_DIS
LIN {X -64.4749,Y 117.1341,Z 184,A 120.2453,B 3.7799,C 0.0601,E1 3.7044,E2 332.8033} C_DIS
LIN {X -67.9345,Y 115.1618,Z 184,A 121.876,B 3.7799,C 0.0629,E1 3.7004,E2 331.1829} C_DIS
LIN {X -71.52,Y 112.9699,Z 184,A 123.6828,B 3.7798,C 0.0654,E1 3.6961,E2 329.3766} C_DIS
LIN {X -74.2653,Y 111.1843,Z 184,A 125.2485,B 3.7798,C 0.0665,E1 3.6925,E2 327.7926} C_DIS
LIN {X -77.8098,Y 108.7333,Z 184,A 127.1141,B 3.7798,C 0.0693,E1 3.6882,E2 325.9261} C_DIS
LIN {X -81.574,Y 105.9393,Z 184,A 129.1344,B 3.7797,C 0.0725,E1 3.6837,E2 323.906} C_DIS
LIN {X -84.7374,Y 103.4257,Z 184,A 130.8858,B 3.7797,C 0.0754,E1 3.6799,E2 322.1534} C_DIS
LIN {X -87.8801,Y 100.7689,Z 184,A 132.7159,B 3.7795,C 0.0781,E1 3.676,E2 320.3168} C_DIS
LIN {X -91.0037,Y 97.9573,Z 184,A 134.5944,B 3.7795,C 0.081,E1 3.6721,E2 318.4304} C_DIS
LIN {X -94.2972,Y 94.791,Z 184,A 136.5597,B 3.7795,C 0.0848,E1 3.6682,E2 316.4657} C_DIS
LIN {X -97.1724,Y 91.8413,Z 184,A 138.4287,B 3.7793,C 0.0877,E1 3.6645,E2 314.5856} C_DIS
LIN {X -100.1353,Y 88.6013,Z 184,A 140.3189,B 3.7793,C 0.0916,E1 3.661,E2 312.6959} C_DIS
LIN {X -102.7282,Y 85.5825,Z 184,A 142.1328,B 3.7792,C 0.0946,E1 3.6577,E2 310.8703} C_DIS
LIN {X -105.412,Y 82.2543,Z 184,A 143.8955,B 3.7791,C 0.099,E1 3.6547,E2 309.1174} C_DIS
LIN {X -107.3924,Y 79.6506,Z 184,A 145.3692,B 3.779,C 0.1017,E1 3.6522,E2 307.6362} C_DIS
LIN {X -109.8367,Y 76.2444,Z 184,A 147.3298,B 3.7789,C 0.1049,E1 3.649,E2 305.6573} C_DIS
LIN {X -112.4397,Y 72.3512,Z 184,A 149.3362,B 3.7788,C 0.1096,E1 3.6459,E2 303.6525} C_DIS
LIN {X -114.2036,Y 69.5341,Z 184,A 150.7861,B 3.7787,C 0.1129,E1 3.6438,E2 302.2007} C_DIS
LIN {X -116.3335,Y 65.9087,Z 184,A 152.7465,B 3.7786,C 0.1165,E1 3.6411,E2 300.2227} C_DIS
LIN {X -118.3972,Y 62.1196,Z 184,A 154.5989,B 3.7784,C 0.121,E1 3.6386,E2 298.3712} C_DIS
LIN {X -120.1581,Y 58.6438,Z 184,A 156.2437,B 3.7783,C 0.1254,E1 3.6366,E2 296.7307} C_DIS
LIN {X -121.8615,Y 55.0158,Z 184,A 158.0131,B 3.7781,C 0.1295,E1 3.6345,E2 294.9565} C_DIS
LIN {X -123.2559,Y 51.8155,Z 184,A 159.7055,B 3.7781,C 0.1324,E1 3.6326,E2 293.2414} C_DIS
LIN {X -125.0002,Y 47.4561,Z 184,A 161.6524,B 3.7778,C 0.138,E1 3.6306,E2 291.304} C_DIS
LIN {X -126.1249,Y 44.381,Z 184,A 163.2947,B 3.7778,C 0.1405,E1 3.6291,E2 289.6337} C_DIS
LIN {X -127.4608,Y 40.3812,Z 184,A 164.9849,B 3.7775,C 0.1459,E1 3.6276,E2 287.9592} C_DIS
LIN {X -128.411,Y 37.2495,Z 184,A 166.44,B 3.7775,C 0.1495,E1 3.6265,E2 286.4988} C_DIS
LIN {X -129.3584,Y 33.8178,Z 184,A 168.1794,B 3.7773,C 0.1526,E1 3.6252,E2 284.7345} C_DIS
LIN {X -130.4407,Y 29.3634,Z 184,A 170.1686,B 3.7771,C 0.1578,E1 3.6239,E2 282.7438} C_DIS
LIN {X -131.3755,Y 24.8472,Z 184,A 172.1544,B 3.7768,C 0.1633,E1 3.6229,E2 280.7583} C_DIS
LIN {X -132.0138,Y 21.2081,Z 184,A 173.7679,B 3.7766,C 0.1675,E1 3.6221,E2 279.1423} C_DIS
LIN {X -132.4888,Y 17.9987,Z 184,A 175.2282,B 3.7765,C 0.1711,E1 3.6215,E2 277.6744} C_DIS
LIN {X -132.891,Y 14.7323,Z 184,A 176.6875,B 3.7763,C 0.1748,E1 3.6211,E2 276.2101} C_DIS
LIN {X -133.2117,Y 11.47,Z 184,A 178.2525,B 3.7762,C 0.178,E1 3.6207,E2 274.6264} C_DIS
LIN {X -133.4965,Y 7.49,Z 184,A -179.8639,B 3.776,C 0.1819,E1 3.6203,E2 272.7227} C_DIS
LIN {X -133.6652,Y 3.2729,Z 184,A -178.1428,B 3.7757,C 0.1875,E1 3.6202,E2 271.0137} C_DIS
LIN {X -133.7026,Y -0.7088,Z 184,A -176.3818,B 3.7755,C 0.192,E1 3.6202,E2 269.247} C_DIS
LIN {X -133.6142,Y -4.9202,Z 184,A -174.4015,B 3.7753,C 0.1962,E1 3.6203,E2 267.2463} C_DIS
LIN {X -133.3947,Y -9.1173,Z 184,A -172.5055,B 3.775,C 0.2008,E1 3.6207,E2 265.3398} C_DIS
LIN {X -133.0606,Y -13.1095,Z 184,A -170.7541,B 3.7748,C 0.2055,E1 3.6211,E2 263.5852} C_DIS
LIN {X -132.5818,Y -17.2895,Z 184,A -169.0172,B 3.7745,C 0.2109,E1 3.6217,E2 261.8576} C_DIS
LIN {X -132.1181,Y -20.5344,Z 184,A -167.5376,B 3.7743,C 0.2144,E1 3.6223,E2 260.3695} C_DIS
LIN {X -131.4481,Y -24.4671,Z 184,A -165.769,B 3.774,C 0.2189,E1 3.6232,E2 258.5947} C_DIS
LIN {X -130.8057,Y -27.6943,Z 184,A -164.1555,B 3.7739,C 0.2217,E1 3.6241,E2 256.9567} C_DIS
LIN {X -129.9202,Y -31.585,Z 184,A -162.5398,B 3.7736,C 0.2269,E1 3.6251,E2 255.3537} C_DIS
LIN {X -129.1016,Y -34.7805,Z 184,A -161.076,B 3.7733,C 0.2304,E1 3.6262,E2 253.8843} C_DIS
LIN {X -128.2138,Y -37.9231,Z 184,A -159.6023,B 3.7731,C 0.2338,E1 3.6273,E2 252.4022} C_DIS
LIN {X -126.9604,Y -41.9278,Z 184,A -157.7567,B 3.7728,C 0.2384,E1 3.6289,E2 250.5515} C_DIS
LIN {X -125.8977,Y -45.0184,Z 184,A -156.3055,B 3.7726,C 0.2418,E1 3.6303,E2 249.0947} C_DIS
LIN {X -124.7156,Y -48.1959,Z 184,A -154.6754,B 3.7724,C 0.2447,E1 3.6319,E2 247.4432} C_DIS
LIN {X -123.2534,Y -51.8214,Z 184,A -153.0339,B 3.7721,C 0.2492,E1 3.6337,E2 245.8067} C_DIS
LIN {X -121.532,Y -55.7395,Z 184,A -151.0205,B 3.7719,C 0.2529,E1 3.636,E2 243.7715} C_DIS
LIN {X -120.156,Y -58.648,Z 184,A -149.7402,B 3.7716,C 0.2569,E1 3.6375,E2 242.5042} C_DIS
LIN {X -118.678,Y -61.5848,Z 184,A -148.3022,B 3.7714,C 0.2602,E1 3.6394,E2 241.0632} C_DIS
LIN {X -117.1381,Y -64.4676,Z 184,A -146.6865,B 3.7712,C 0.2624,E1 3.6415,E2 239.421} C_DIS
LIN {X -115.1496,Y -67.9554,Z 184,A -145.019,B 3.7709,C 0.2668,E1 3.6439,E2 237.7607} C_DIS
LIN {X -112.964,Y -71.5294,Z 184,A -143.1918,B 3.7707,C 0.2709,E1 3.6466,E2 235.9302} C_DIS
LIN {X -111.1759,Y -74.2779,Z 184,A -141.6035,B 3.7705,C 0.273,E1 3.6491,E2 234.3191} C_DIS
LIN {X -108.5831,Y -78.0198,Z 184,A -139.652,B 3.7702,C 0.2774,E1 3.6522,E2 232.3681} C_DIS
LIN {X -106.1224,Y -81.3348,Z 184,A -137.8531,B 3.7699,C 0.2811,E1 3.6552,E2 230.5659} C_DIS
LIN {X -103.5805,Y -84.548,Z 184,A -136.0335,B 3.7696,C 0.2845,E1 3.6584,E2 228.7388} C_DIS
LIN {X -100.7077,Y -87.9503,Z 184,A -134.0772,B 3.7694,C 0.2882,E1 3.662,E2 226.7767} C_DIS
LIN {X -97.9568,Y -91.0043,Z 184,A -132.2555,B 3.7691,C 0.2913,E1 3.6654,E2 224.9478} C_DIS
LIN {X -95.1253,Y -93.9607,Z 184,A -130.42,B 3.7689,C 0.2942,E1 3.669,E2 223.1022} C_DIS
LIN {X -92.204,Y -96.8285,Z 184,A -128.6577,B 3.7686,C 0.2975,E1 3.6726,E2 221.3391} C_DIS
LIN {X -89.1819,Y -99.6186,Z 184,A -126.842,B 3.7684,C 0.3003,E1 3.6763,E2 219.5168} C_DIS
LIN {X -85.8157,Y -102.5328,Z 184,A -124.8802,B 3.7682,C 0.3033,E1 3.6805,E2 217.5484} C_DIS
LIN {X -82.3544,Y -105.3334,Z 184,A -122.9905,B 3.7679,C 0.3066,E1 3.6847,E2 215.6611} C_DIS
LIN {X -79.641,Y -107.3995,Z 184,A -121.514,B 3.7677,C 0.3088,E1 3.688,E2 214.1829} C_DIS
LIN {X -76.9851,Y -109.3188,Z 184,A -119.9461,B 3.7677,C 0.3099,E1 3.6916,E2 212.594} C_DIS
LIN {X -73.6908,Y -111.5661,Z 184,A -118.3447,B 3.7674,C 0.3131,E1 3.6953,E2 211.0064} C_DIS
LIN {X -70.7513,Y -113.4529,Z 184,A -116.7701,B 3.7673,C 0.3147,E1 3.699,E2 209.4218} C_DIS
LIN {X -67.3351,Y -115.5138,Z 184,A -114.9304,B 3.7671,C 0.316,E1 3.7035,E2 207.5654} C_DIS
LIN {X -63.8494,Y -117.4759,Z 184,A -113.2684,B 3.7669,C 0.3185,E1 3.7075,E2 205.9099} C_DIS
LIN {X -60.9331,Y -119.0125,Z 184,A -111.8993,B 3.7668,C 0.3205,E1 3.7109,E2 204.5462} C_DIS
LIN {X -57.8064,Y -120.562,Z 184,A -110.3788,B 3.7666,C 0.322,E1 3.7147,E2 203.0223} C_DIS
LIN {X -54.6143,Y -122.0411,Z 184,A -108.7722,B 3.7666,C 0.3228,E1 3.7189,E2 201.4027} C_DIS
LIN {X -51.1724,Y -123.5245,Z 184,A -107.2177,B 3.7664,C 0.3248,E1 3.7228,E2 199.8547} C_DIS
LIN {X -47.4723,Y -124.9941,Z 184,A -105.481,B 3.7663,C 0.3261,E1 3.7274,E2 198.1137} C_DIS
LIN {X -44.3802,Y -126.1251,Z 184,A -103.8695,B 3.7663,C 0.3257,E1 3.7317,E2 196.4762} C_DIS
LIN {X -39.8186,Y -127.6393,Z 184,A -101.8828,B 3.7661,C 0.3278,E1 3.7369,E2 194.4983} C_DIS
LIN {X -35.6611,Y -128.8612,Z 184,A -100.084,B 3.766,C 0.3294,E1 3.7418,E2 192.7065} C_DIS
LIN {X -31.5909,Y -129.9188,Z 184,A -98.1741,B 3.766,C 0.3295,E1 3.747,E2 190.7823} C_DIS
LIN {X -26.993,Y -130.9516,Z 184,A -96.2122,B 3.7659,C 0.3309,E1 3.7523,E2 188.8271} C_DIS
LIN {X -23.5624,Y -131.6117,Z 184,A -94.761,B 3.7658,C 0.3318,E1 3.7563,E2 187.3813} C_DIS
LIN {X -20.5454,Y -132.1164,Z 184,A -93.4436,B 3.7658,C 0.3322,E1 3.7599,E2 186.0626} C_DIS
LIN {X -17.3027,Y -132.5801,Z 184,A -92.0094,B 3.7658,C 0.3322,E1 3.7639,E2 184.624} C_DIS
LIN {X -13.1027,Y -133.0612,Z 184,A -90.1654,B 3.7658,C 0.3322,E1 3.7691,E2 182.775} C_DIS
LIN {X -9.1356,Y -133.3933,Z 184,A -88.5318,B 3.7657,C 0.333,E1 3.7736,E2 181.1501} C_DIS
LIN {X -4.937,Y -133.6136,Z 184,A -86.5832,B 3.7657,C 0.3317,E1 3.7791,E2 179.1817} C_DIS
LIN {X -0.7338,Y -133.7025,Z 184,A -84.9023,B 3.7657,C 0.3325,E1 3.7837,E2 177.5156} C_DIS
LIN {X -0.7338,Y -133.7025,Z 184,A -84.9023,B 3.7657,C 0.3325,E1 3.7837,E2 177.5156} C_DIS
Enddeposition()
LIN {X 0.9672,Y -134.6001,Z 184,A -84.8735,B 3.7649,C 0.3405,E1 3.7834,E2 177.6078} C_DIS
Startdeposition()
$VEL.CP = VEL_PRINT
LIN {X -4.1513,Y -134.542,Z 184,A -86.9058,B 3.765,C 0.3394,E1 3.7778,E2 179.6223} C_DIS
LIN {X -7.3856,Y -134.404,Z 184,A -88.4495,B 3.7649,C 0.3409,E1 3.7734,E2 181.1879} C_DIS
LIN {X -11.2036,Y -134.1383,Z 184,A -89.9937,B 3.7649,C 0.34,E1 3.7691,E2 182.7219} C_DIS
LIN {X -16.2808,Y -133.6174,Z 184,A -92.0926,B 3.7651,C 0.3391,E1 3.7633,E2 184.8122} C_DIS
LIN {X -19.1856,Y -133.2309,Z 184,A -93.4009,B 3.7651,C 0.3393,E1 3.7597,E2 186.1288} C_DIS
LIN {X -22.7846,Y -132.6643,Z 184,A -95.0971,B 3.765,C 0.34,E1 3.7549,E2 187.8442} C_DIS
LIN {X -26.9312,Y -131.8835,Z 184,A -96.755,B 3.7651,C 0.3382,E1 3.7504,E2 189.485} C_DIS
LIN {X -30.1863,Y -131.1768,Z 184,A -98.206,B 3.7651,C 0.3377,E1 3.7465,E2 190.9407} C_DIS
LIN {X -33.3941,Y -130.3972,Z 184,A -99.5807,B 3.7653,C 0.3367,E1 3.7427,E2 192.3119} C_DIS
LIN {X -36.8141,Y -129.4742,Z 184,A -101.2557,B 3.7653,C 0.3371,E1 3.7382,E2 194.0088} C_DIS
LIN {X -43.7715,Y -127.2896,Z 184,A -104.0688,B 3.7656,C 0.3327,E1 3.7308,E2 196.7853} C_DIS
LIN {X -46.076,Y -126.474,Z 184,A -105.4352,B 3.7655,C 0.3342,E1 3.7271,E2 198.1937} C_DIS
LIN {X -50.5388,Y -124.7572,Z 184,A -107.4188,B 3.7657,C 0.332,E1 3.7219,E2 200.1711} C_DIS
LIN {X -53.7136,Y -123.4237,Z 184,A -108.8664,B 3.7658,C 0.3305,E1 3.7182,E2 201.6165} C_DIS
LIN {X -56.729,Y -122.0669,Z 184,A -110.2722,B 3.766,C 0.329,E1 3.7146,E2 203.0223} C_DIS
LIN {X -59.7256,Y -120.6289,Z 184,A -111.7553,B 3.766,C 0.3279,E1 3.7109,E2 204.5144} C_DIS
LIN {X -63.2188,Y -118.8375,Z 184,A -113.5137,B 3.7662,C 0.3265,E1 3.7065,E2 206.284} C_DIS
LIN {X -67.9508,Y -116.1971,Z 184,A -115.6258,B 3.7665,C 0.3223,E1 3.7014,E2 208.3715} C_DIS
LIN {X -70.7581,Y -114.5097,Z 184,A -117.2562,B 3.7665,C 0.322,E1 3.6975,E2 210.0321} C_DIS
LIN {X -74.2239,Y -112.2937,Z 184,A -119.0222,B 3.7668,C 0.3196,E1 3.6933,E2 211.8001} C_DIS
LIN {X -77.3535,Y -110.1613,Z 184,A -120.7359,B 3.7669,C 0.3178,E1 3.6894,E2 213.5267} C_DIS
LIN {X -80.7552,Y -107.6929,Z 184,A -122.5918,B 3.7671,C 0.3155,E1 3.6852,E2 215.3911} C_DIS
LIN {X -84.3792,Y -104.8769,Z 184,A -124.5276,B 3.7674,C 0.3121,E1 3.6809,E2 217.3244} C_DIS
LIN {X -87.6481,Y -102.161,Z 184,A -126.3904,B 3.7676,C 0.3094,E1 3.6769,E2 219.194} C_DIS
LIN {X -90.8538,Y -99.3211,Z 184,A -128.2553,B 3.7679,C 0.3063,E1 3.6731,E2 221.0639} C_DIS
LIN {X -94.0415,Y -96.3082,Z 184,A -130.1842,B 3.7681,C 0.3032,E1 3.6692,E2 223.0004} C_DIS
LIN {X -97.1281,Y -93.1943,Z 184,A -132.088,B 3.7684,C 0.2998,E1 3.6654,E2 224.9086} C_DIS
LIN {X -100.2479,Y -89.8295,Z 184,A -134.082,B 3.7687,C 0.2962,E1 3.6617,E2 226.9073} C_DIS
LIN {X -103.4406,Y -86.1346,Z 184,A -136.2508,B 3.769,C 0.2924,E1 3.6577,E2 229.0871} C_DIS
LIN {X -106.143,Y -82.7818,Z 184,A -138.1201,B 3.7692,C 0.2887,E1 3.6545,E2 230.9606} C_DIS
LIN {X -108.7878,Y -79.2738,Z 184,A -140.0402,B 3.7695,C 0.2848,E1 3.6513,E2 232.8864} C_DIS
LIN {X -111.2372,Y -75.7987,Z 184,A -141.9131,B 3.7698,C 0.2811,E1 3.6483,E2 234.7666} C_DIS
LIN {X -113.55,Y -72.2876,Z 184,A -143.7791,B 3.7701,C 0.2774,E1 3.6454,E2 236.6417} C_DIS
LIN {X -115.8127,Y -68.6042,Z 184,A -145.8335,B 3.7703,C 0.2742,E1 3.6424,E2 238.7222} C_DIS
LIN {X -117.6401,Y -65.4206,Z 184,A -147.2863,B 3.7706,C 0.2698,E1 3.6405,E2 240.1608} C_DIS
LIN {X -119.9179,Y -61.1404,Z 184,A -149.3642,B 3.771,C 0.2648,E1 3.6378,E2 242.2396} C_DIS
LIN {X -121.4064,Y -58.1288,Z 184,A -150.8267,B 3.7712,C 0.2614,E1 3.636,E2 243.7055} C_DIS
LIN {X -122.8241,Y -55.07,Z 184,A -152.3595,B 3.7714,C 0.2583,E1 3.6342,E2 245.2499} C_DIS
LIN {X -124.3433,Y -51.5492,Z 184,A -153.967,B 3.7717,C 0.254,E1 3.6324,E2 246.8536} C_DIS
LIN {X -125.6219,Y -48.3508,Z 184,A -156.1042,B 3.7717,C 0.2537,E1 3.6302,E2 249.0735} C_DIS
LIN {X -127.2307,Y -43.9415,Z 184,A -157.6235,B 3.7723,C 0.2459,E1 3.6289,E2 250.5325} C_DIS
LIN {X -128.6123,Y -39.7176,Z 184,A -159.5824,B 3.7726,C 0.2412,E1 3.6272,E2 252.4988} C_DIS
LIN {X -129.6685,Y -36.1194,Z 184,A -161.5632,B 3.7727,C 0.2389,E1 3.6256,E2 254.5263} C_DIS
LIN {X -130.5915,Y -32.6284,Z 184,A -162.6806,B 3.7731,C 0.2326,E1 3.6249,E2 255.5909} C_DIS
LIN {X -131.2458,Y -29.8841,Z 184,A -164.0388,B 3.7733,C 0.2301,E1 3.624,E2 256.9679} C_DIS
LIN {X -131.9313,Y -26.6961,Z 184,A -165.502,B 3.7735,C 0.2266,E1 3.6232,E2 258.4397} C_DIS
LIN {X -132.6291,Y -22.9913,Z 184,A -167.2586,B 3.7737,C 0.223,E1 3.6223,E2 260.2142} C_DIS
LIN {X -133.2678,Y -18.928,Z 184,A -168.9345,B 3.774,C 0.2177,E1 3.6216,E2 261.8797} C_DIS
LIN {X -133.688,Y -15.6893,Z 184,A -170.5039,B 3.7742,C 0.2147,E1 3.6211,E2 263.4703} C_DIS
LIN {X -134.1147,Y -11.4831,Z 184,A -172.3489,B 3.7744,C 0.2099,E1 3.6206,E2 265.3197} C_DIS
LIN {X -134.3959,Y -7.5412,Z 184,A -174.1657,B 3.7747,C 0.2058,E1 3.6203,E2 267.1521} C_DIS
LIN {X -134.5627,Y -3.4068,Z 184,A -175.8188,B 3.775,C 0.2003,E1 3.6201,E2 268.7907} C_DIS
LIN {X -134.6056,Y 0.2889,Z 184,A -177.5362,B 3.7752,C 0.1966,E1 3.6201,E2 270.5247} C_DIS
LIN {X -134.5502,Y 3.8536,Z 184,A -179.0915,B 3.7754,C 0.1925,E1 3.6201,E2 272.0835} C_DIS
LIN {X -134.3879,Y 7.6716,Z 184,A 179.0889,B 3.7756,C 0.1888,E1 3.6204,E2 273.9257} C_DIS
LIN {X -134.0792,Y 11.9029,Z 184,A 177.2292,B 3.7758,C 0.184,E1 3.6209,E2 275.7907} C_DIS
LIN {X -133.6649,Y 15.8826,Z 184,A 175.5728,B 3.776,C 0.179,E1 3.6214,E2 277.44} C_DIS
LIN {X -133.1822,Y 19.5265,Z 184,A 173.8581,B 3.7762,C 0.1754,E1 3.622,E2 279.1719} C_DIS
LIN {X -132.5137,Y 23.6358,Z 184,A 171.7084,B 3.7763,C 0.1723,E1 3.6231,E2 281.3661} C_DIS
LIN {X -131.7961,Y 27.3605,Z 184,A 169.8865,B 3.7765,C 0.1688,E1 3.6241,E2 283.2118} C_DIS
LIN {X -130.834,Y 31.6384,Z 184,A 168.4389,B 3.7768,C 0.1616,E1 3.625,E2 284.6074} C_DIS
LIN {X -129.6515,Y 36.1801,Z 184,A 166.3403,B 3.777,C 0.1567,E1 3.6266,E2 286.7166} C_DIS
LIN {X -128.5177,Y 40.0267,Z 184,A 164.62,B 3.7772,C 0.1521,E1 3.628,E2 288.4373} C_DIS
LIN {X -126.943,Y 44.7715,Z 184,A 162.4576,B 3.7774,C 0.1466,E1 3.6299,E2 290.6023} C_DIS
LIN {X -125.9514,Y 47.4848,Z 184,A 161.1031,B 3.7775,C 0.144,E1 3.6312,E2 291.9707} C_DIS
LIN {X -124.6653,Y 50.7666,Z 184,A 159.5881,B 3.7777,C 0.1401,E1 3.6328,E2 293.4864} C_DIS
LIN {X -123.1973,Y 54.2355,Z 184,A 157.6843,B 3.7777,C 0.1375,E1 3.635,E2 295.4252} C_DIS
LIN {X -121.3379,Y 58.2722,Z 184,A 155.9854,B 3.778,C 0.1317,E1 3.6369,E2 297.0992} C_DIS
LIN {X -119.6878,Y 61.5923,Z 184,A 154.2077,B 3.778,C 0.1288,E1 3.6392,E2 298.8998} C_DIS
LIN {X -117.455,Y 65.7523,Z 184,A 152.174,B 3.7782,C 0.124,E1 3.6419,E2 300.9347} C_DIS
LIN {X -115.2686,Y 69.5138,Z 184,A 150.2573,B 3.7784,C 0.1198,E1 3.6447,E2 302.8577} C_DIS
LIN {X -111.4982,Y 75.4132,Z 184,A 147.1933,B 3.7786,C 0.1133,E1 3.6494,E2 305.9293} C_DIS
LIN {X -109.1383,Y 78.7901,Z 184,A 145.3956,B 3.7786,C 0.1095,E1 3.6523,E2 307.7309} C_DIS
LIN {X -106.8752,Y 81.8333,Z 184,A 143.2873,B 3.7787,C 0.1086,E1 3.6559,E2 309.8967} C_DIS
LIN {X -104.1958,Y 85.2187,Z 184,A 141.9186,B 3.7789,C 0.102,E1 3.6582,E2 311.2082} C_DIS
LIN {X -101.5132,Y 88.3973,Z 184,A 139.7519,B 3.7789,C 0.1005,E1 3.6623,E2 313.4206} C_DIS
LIN {X -99.244,Y 90.9376,Z 184,A 138.8432,B 3.7791,C 0.0945,E1 3.6639,E2 314.2638} C_DIS
LIN {X -92.5772,Y 97.7166,Z 184,A 134.3514,B 3.7792,C 0.0891,E1 3.6728,E2 318.8056} C_DIS
LIN {X -89.4321,Y 100.6033,Z 184,A 132.4451,B 3.7792,C 0.0862,E1 3.6768,E2 320.721} C_DIS
LIN {X -84.2709,Y 104.9642,Z 184,A 129.2565,B 3.7794,C 0.083,E1 3.6837,E2 323.9444} C_DIS
LIN {X -81.5152,Y 107.117,Z 184,A 127.6005,B 3.7794,C 0.0816,E1 3.6874,E2 325.6189} C_DIS
LIN {X -78.0232,Y 109.6881,Z 184,A 125.7251,B 3.7794,C 0.0788,E1 3.6917,E2 327.4965} C_DIS
LIN {X -74.5709,Y 112.0634,Z 184,A 124.3603,B 3.7796,C 0.0735,E1 3.6947,E2 328.8107} C_DIS
LIN {X -70.9637,Y 114.3817,Z 184,A 122.4149,B 3.7796,C 0.0716,E1 3.6994,E2 330.769} C_DIS
LIN {X -67.1634,Y 116.6541,Z 184,A 120.5354,B 3.7796,C 0.069,E1 3.7039,E2 332.6465} C_DIS
LIN {X -63.6283,Y 118.6189,Z 184,A 118.5783,B 3.7796,C 0.0683,E1 3.7088,E2 334.6301} C_DIS
LIN {X -59.5804,Y 120.7005,Z 184,A 116.8322,B 3.7797,C 0.0648,E1 3.7131,E2 336.3523} C_DIS
LIN {X -55.9062,Y 122.4474,Z 184,A 115.1387,B 3.7797,C 0.0626,E1 3.7173,E2 338.0402} C_DIS
LIN {X -50.6454,Y 124.7142,Z 184,A 111.9029,B 3.7797,C 0.0654,E1 3.7259,E2 341.3679} C_DIS
LIN {X -45.4269,Y 126.708,Z 184,A 110.2034,B 3.7798,C 0.0587,E1 3.7302,E2 342.9865} C_DIS
LIN {X -39.0182,Y 128.8263,Z 184,A 107.4178,B 3.7798,C 0.0558,E1 3.7376,E2 345.76} C_DIS
LIN {X -36.204,Y 129.6448,Z 184,A 106.0592,B 3.7798,C 0.0558,E1 3.7412,E2 347.1309} C_DIS
LIN {X -32.6191,Y 130.5939,Z 184,A 104.3723,B 3.7798,C 0.0555,E1 3.7458,E2 348.8298} C_DIS
LIN {X -28.4467,Y 131.5649,Z 184,A 102.6115,B 3.7798,C 0.0541,E1 3.7506,E2 350.5821} C_DIS
LIN {X -24.2227,Y 132.4087,Z 184,A 100.7013,B 3.7798,C 0.0538,E1 3.7559,E2 352.5004} C_DIS
LIN {X -20.6246,Y 133.0157,Z 184,A 99.2092,B 3.7799,C 0.0528,E1 3.76,E2 353.9845} C_DIS
LIN {X -16.5359,Y 133.587,Z 184,A 97.1398,B 3.7799,C 0.0547,E1 3.7658,E2 356.0897} C_DIS
LIN {X -13.1306,Y 133.9636,Z 184,A 96.21,B 3.7799,C 0.0504,E1 3.7682,E2 356.9565} C_DIS
LIN {X -9.7374,Y 134.2526,Z 184,A 94.5737,B 3.7799,C 0.0516,E1 3.7728,E2 358.6141} C_DIS
LIN {X -6.1174,Y 134.4678,Z 184,A 93.012,B 3.7799,C 0.0516,E1 3.7772,E2 360.1774} C_DIS
LIN {X -1.7956,Y 134.5941,Z 184,A 91.0431,B 3.7799,C 0.0527,E1 3.7827,E2 362.1606} C_DIS
LIN {X 2.4918,Y 134.5826,Z 184,A 89.3674,B 3.7799,C 0.0518,E1 3.7874,E2 363.8179} C_DIS
LIN {X 6.496,Y 134.4487,Z 184,A 87.6121,B 3.7799,C 0.0525,E1 3.7923,E2 365.5784} C_DIS
LIN {X 10.3346,Y 134.209,Z 184,A 85.7777,B 3.7799,C 0.0546,E1 3.7975,E2 367.4354} C_DIS
LIN {X 14.2174,Y 133.8524,Z 184,A 84.3494,B 3.7799,C 0.0533,E1 3.8013,E2 368.8358} C_DIS
LIN {X 17.5819,Y 133.452,Z 184,A 82.9297,B 3.7799,C 0.0537,E1 3.8053,E2 370.2524} C_DIS
LIN {X 21.0457,Y 132.9505,Z 184,A 81.4479,B 3.7799,C 0.0544,E1 3.8094,E2 371.7328} C_DIS
LIN {X 24.9202,Y 132.2787,Z 184,A 79.7409,B 3.7799,C 0.0557,E1 3.8141,E2 373.4432} C_DIS
LIN {X 28.3882,Y 131.5775,Z 184,A 78.2872,B 3.7799,C 0.0563,E1 3.818,E2 374.8903} C_DIS
LIN {X 32.0952,Y 130.7239,Z 184,A 76.7252,B 3.7799,C 0.057,E1 3.8223,E2 376.4451} C_DIS
LIN {X 35.0693,Y 129.957,Z 184,A 75.449,B 3.7799,C 0.0577,E1 3.8257,E2 377.7173} C_DIS
LIN {X 40.8813,Y 128.2467,Z 184,A 73.1559,B 3.7799,C 0.0575,E1 3.8318,E2 379.9758} C_DIS
LIN {X 43.7349,Y 127.3023,Z 184,A 71.49,B 3.7798,C 0.0622,E1 3.8363,E2 381.6875} C_DIS
LIN {X 47.7766,Y 125.8421,Z 184,A 69.832,B 3.7798,C 0.0626,E1 3.8406,E2 383.3249} C_DIS
LIN {X 50.2523,Y 124.8726,Z 184,A 68.6543,B 3.7798,C 0.0643,E1 3.8436,E2 384.5078} C_DIS
LIN {X 53.4152,Y 123.5527,Z 184,A 67.2163,B 3.7797,C 0.0658,E1 3.8473,E2 385.9431} C_DIS
LIN {X 56.8988,Y 121.9884,Z 184,A 65.6652,B 3.7797,C 0.0671,E1 3.8513,E2 387.4852} C_DIS
LIN {X 60.1167,Y 120.436,Z 184,A 64.1943,B 3.7797,C 0.0687,E1 3.8549,E2 388.9501} C_DIS
LIN {X 62.5832,Y 119.1712,Z 184,A 62.5672,B 3.7795,C 0.0745,E1 3.8591,E2 390.6301} C_DIS
LIN {X 66.2601,Y 117.1696,Z 184,A 61.4441,B 3.7796,C 0.0708,E1 3.8617,E2 391.6749} C_DIS
LIN {X 70.3752,Y 114.7446,Z 184,A 59.2236,B 3.7796,C 0.0757,E1 3.867,E2 393.9177} C_DIS
LIN {X 73.8775,Y 112.5217,Z 184,A 57.4236,B 3.7795,C 0.0788,E1 3.8713,E2 395.7218} C_DIS
LIN {X 77.7434,Y 109.8863,Z 184,A 55.485,B 3.7794,C 0.0816,E1 3.8757,E2 397.6541} C_DIS
LIN {X 81.183,Y 107.37,Z 184,A 53.7361,B 3.7794,C 0.0842,E1 3.8796,E2 399.3954} C_DIS
LIN {X 84.7191,Y 104.6027,Z 184,A 51.8762,B 3.7793,C 0.0871,E1 3.8837,E2 401.2492} C_DIS
LIN {X 88.1237,Y 101.7514,Z 184,A 49.9926,B 3.7792,C 0.0906,E1 3.8877,E2 403.1323} C_DIS
LIN {X 92.1043,Y 98.1628,Z 184,A 47.7534,B 3.7791,C 0.0946,E1 3.8923,E2 405.3668} C_DIS
LIN {X 95.3894,Y 94.973,Z 184,A 45.8004,B 3.779,C 0.0986,E1 3.8961,E2 407.3205} C_DIS
LIN {X 98.2557,Y 92.0051,Z 184,A 44.1508,B 3.779,C 0.1012,E1 3.8993,E2 408.9576} C_DIS
LIN {X 101.2458,Y 88.7037,Z 184,A 42.3148,B 3.7788,C 0.1046,E1 3.9027,E2 410.7868} C_DIS
LIN {X 104.0781,Y 85.3627,Z 184,A 40.5294,B 3.7788,C 0.1079,E1 3.9059,E2 412.5632} C_DIS
LIN {X 106.7741,Y 81.9655,Z 184,A 38.7156,B 3.7786,C 0.1118,E1 3.909,E2 414.3735} C_DIS
LIN {X 109.4352,Y 78.3769,Z 184,A 36.876,B 3.7786,C 0.1155,E1 3.912,E2 416.2062} C_DIS
LIN {X 111.8812,Y 74.8438,Z 184,A 35.122,B 3.7784,C 0.119,E1 3.9147,E2 417.9517} C_DIS
LIN {X 114.1621,Y 71.3166,Z 184,A 33.4587,B 3.7784,C 0.122,E1 3.9172,E2 419.6005} C_DIS
LIN {X 116.0909,Y 68.1315,Z 184,A 31.8494,B 3.7782,C 0.1261,E1 3.9195,E2 421.2132} C_DIS
LIN {X 118.2883,Y 64.2412,Z 184,A 29.9861,B 3.778,C 0.1304,E1 3.922,E2 423.0727} C_DIS
LIN {X 120.0794,Y 60.8231,Z 184,A 28.485,B 3.778,C 0.1331,E1 3.9239,E2 424.5571} C_DIS
LIN {X 121.7552,Y 57.3987,Z 184,A 26.9264,B 3.7778,C 0.1365,E1 3.9258,E2 426.1086} C_DIS
LIN {X 123.4779,Y 53.5884,Z 184,A 25.1611,B 3.7776,C 0.141,E1 3.9278,E2 427.8729} C_DIS
LIN {X 124.9651,Y 50.0228,Z 184,A 23.6363,B 3.7776,C 0.144,E1 3.9294,E2 429.3838} C_DIS
LIN {X 126.4273,Y 46.2057,Z 184,A 21.729,B 3.7773,C 0.1504,E1 3.9313,E2 431.3123} C_DIS
LIN {X 128.2252,Y 40.9485,Z 184,A 19.6846,B 3.7772,C 0.1532,E1 3.9331,E2 433.3187} C_DIS
LIN {X 129.2851,Y 37.4698,Z 184,A 18.1608,B 3.777,C 0.1572,E1 3.9343,E2 434.8404} C_DIS
LIN {X 130.4124,Y 33.3343,Z 184,A 16.3807,B 3.7768,C 0.1617,E1 3.9356,E2 436.6161} C_DIS
LIN {X 131.2707,Y 29.7751,Z 184,A 14.9009,B 3.7767,C 0.1651,E1 3.9365,E2 438.087} C_DIS
LIN {X 132.0558,Y 26.0842,Z 184,A 13.2467,B 3.7764,C 0.1701,E1 3.9374,E2 439.7482} C_DIS
LIN {X 132.7741,Y 22.1263,Z 184,A 11.7216,B 3.7764,C 0.1728,E1 3.9381,E2 441.2512} C_DIS
LIN {X 133.343,Y 18.4012,Z 184,A 10.203,B 3.7762,C 0.1763,E1 3.9388,E2 442.7603} C_DIS
LIN {X 133.8582,Y 14.1634,Z 184,A 8.3655,B 3.7759,C 0.1816,E1 3.9393,E2 444.6013} C_DIS
LIN {X 134.3152,Y 8.8506,Z 184,A 6.1271,B 3.7756,C 0.1877,E1 3.9398,E2 446.8374} C_DIS
LIN {X 134.5138,Y 4.9721,Z 184,A 4.5712,B 3.7754,C 0.1912,E1 3.94,E2 448.3823} C_DIS
LIN {X 134.6049,Y 0.4284,Z 184,A 2.7178,B 3.7752,C 0.1958,E1 3.94,E2 450.227} C_DIS
LIN {X 134.5312,Y -4.5161,Z 184,A 0.6347,B 3.7749,C 0.2015,E1 3.94,E2 452.3089} C_DIS
LIN {X 134.345,Y -8.3668,Z 184,A -0.8529,B 3.7747,C 0.2044,E1 3.9397,E2 453.7785} C_DIS
LIN {X 134.0696,Y -12.0153,Z 184,A -2.5675,B 3.7744,C 0.2106,E1 3.9393,E2 455.5139} C_DIS
LIN {X 133.6109,Y -16.3352,Z 184,A -4.1586,B 3.7743,C 0.2129,E1 3.9388,E2 457.0742} C_DIS
LIN {X 133.0646,Y -20.3086,Z 184,A -5.8107,B 3.774,C 0.217,E1 3.9382,E2 458.7206} C_DIS
LIN {X 132.4288,Y -24.1107,Z 184,A -7.4462,B 3.7738,C 0.2216,E1 3.9374,E2 460.3567} C_DIS
LIN {X 131.603,Y -28.2701,Z 184,A -9.1153,B 3.7736,C 0.225,E1 3.9364,E2 462.0102} C_DIS
LIN {X 130.6922,Y -32.2268,Z 184,A -10.8678,B 3.7733,C 0.2301,E1 3.9353,E2 463.7671} C_DIS
LIN {X 129.7055,Y -35.987,Z 184,A -12.3828,B 3.7731,C 0.2331,E1 3.9342,E2 465.2659} C_DIS
LIN {X 128.6392,Y -39.6297,Z 184,A -13.9125,B 3.7729,C 0.2365,E1 3.933,E2 466.786} C_DIS
LIN {X 125.9589,Y -47.4646,Z 184,A -17.0703,B 3.7725,C 0.2419,E1 3.9302,E2 469.9006} C_DIS
LIN {X 124.1845,Y -51.9296,Z 184,A -19.256,B 3.7721,C 0.2489,E1 3.9279,E2 472.1057} C_DIS
LIN {X 122.7678,Y -55.1959,Z 184,A -20.7278,B 3.7719,C 0.2524,E1 3.9262,E2 473.5732} C_DIS
LIN {X 121.3768,Y -58.1907,Z 184,A -22.1096,B 3.7716,C 0.2557,E1 3.9245,E2 474.9532} C_DIS
LIN {X 119.8536,Y -61.2668,Z 184,A -23.8705,B 3.7711,C 0.2628,E1 3.9223,E2 476.753} C_DIS
LIN {X 118.0637,Y -64.653,Z 184,A -25.1792,B 3.7711,C 0.2634,E1 3.9206,E2 478.0226} C_DIS
LIN {X 116.0338,Y -68.2287,Z 184,A -26.879,B 3.7708,C 0.2672,E1 3.9182,E2 479.7175} C_DIS
LIN {X 113.7312,Y -72.0017,Z 184,A -28.6656,B 3.7706,C 0.2707,E1 3.9156,E2 481.4937} C_DIS
LIN {X 111.2903,Y -75.7204,Z 184,A -30.8202,B 3.77,C 0.2781,E1 3.9122,E2 483.6829} C_DIS
LIN {X 109.1101,Y -78.8291,Z 184,A -32.0593,B 3.77,C 0.2778,E1 3.9102,E2 484.8756} C_DIS
LIN {X 106.5838,Y -82.2131,Z 184,A -33.8619,B 3.7698,C 0.282,E1 3.9072,E2 486.6804} C_DIS
LIN {X 103.7997,Y -85.701,Z 184,A -35.6949,B 3.7695,C 0.2856,E1 3.904,E2 488.5064} C_DIS
LIN {X 100.8806,Y -89.1185,Z 184,A -37.5802,B 3.7692,C 0.2895,E1 3.9005,E2 490.3898} C_DIS
LIN {X 97.6496,Y -92.6482,Z 184,A -39.6118,B 3.7689,C 0.2938,E1 3.8967,E2 492.4225} C_DIS
LIN {X 95.0683,Y -95.2947,Z 184,A -41.0743,B 3.7687,C 0.2959,E1 3.8938,E2 493.8722} C_DIS
LIN {X 91.7359,Y -98.5065,Z 184,A -42.9663,B 3.7684,C 0.2991,E1 3.89,E2 495.7558} C_DIS
LIN {X 89.222,Y -100.789,Z 184,A -44.3573,B 3.7683,C 0.3014,E1 3.8871,E2 497.141} C_DIS
LIN {X 85.7464,Y -103.762,Z 184,A -46.0834,B 3.7681,C 0.3028,E1 3.8835,E2 498.8405} C_DIS
LIN {X 83.1047,Y -105.8896,Z 184,A -47.6787,B 3.7678,C 0.307,E1 3.8799,E2 500.4564} C_DIS
LIN {X 79.6375,Y -108.5213,Z 184,A -49.5552,B 3.7675,C 0.3106,E1 3.8757,E2 502.3373} C_DIS
LIN {X 75.9337,Y -111.1447,Z 184,A -51.3877,B 3.7673,C 0.3129,E1 3.8716,E2 504.1586} C_DIS
LIN {X 72.063,Y -113.6925,Z 184,A -53.1328,B 3.7673,C 0.3138,E1 3.8675,E2 505.8762} C_DIS
LIN {X 69.9727,Y -114.9911,Z 184,A -55.048,B 3.7664,C 0.3242,E1 3.8627,E2 507.9027} C_DIS
LIN {X 64.7233,Y -118.0253,Z 184,A -57.2111,B 3.7664,C 0.3239,E1 3.8575,E2 510.0148} C_DIS
LIN {X 61.2498,Y -119.8622,Z 184,A -58.1734,B 3.7668,C 0.3192,E1 3.8554,E2 510.8873} C_DIS
LIN {X 57.8232,Y -121.5523,Z 184,A -59.9792,B 3.7665,C 0.3232,E1 3.8508,E2 512.7174} C_DIS
LIN {X 54.9136,Y -122.8941,Z 184,A -61.3413,B 3.7663,C 0.3249,E1 3.8473,E2 514.0802} C_DIS
LIN {X 51.599,Y -124.3225,Z 184,A -62.8776,B 3.7661,C 0.3268,E1 3.8433,E2 515.6176} C_DIS
LIN {X 48.2923,Y -125.6447,Z 184,A -64.3336,B 3.7661,C 0.328,E1 3.8396,E2 517.067} C_DIS
LIN {X 45.6901,Y -126.6132,Z 184,A -65.5374,B 3.7659,C 0.3295,E1 3.8364,E2 518.2744} C_DIS
LIN {X 42.1439,Y -127.838,Z 184,A -67.0609,B 3.7659,C 0.3304,E1 3.8324,E2 519.7896} C_DIS
LIN {X 39.0682,Y -128.811,Z 184,A -68.4658,B 3.7657,C 0.3321,E1 3.8286,E2 521.1995} C_DIS
LIN {X 34.9534,Y -129.9879,Z 184,A -70.2629,B 3.7656,C 0.3335,E1 3.8238,E2 522.9945} C_DIS
LIN {X 31.3875,Y -130.8945,Z 184,A -71.7413,B 3.7656,C 0.3339,E1 3.8198,E2 524.4626} C_DIS
LIN {X 28.0974,Y -131.6403,Z 184,A -73.1893,B 3.7654,C 0.3351,E1 3.8158,E2 525.9131} C_DIS
LIN {X 23.9556,Y -132.4565,Z 184,A -75.0181,B 3.7653,C 0.3366,E1 3.8108,E2 527.7471} C_DIS
LIN {X 20.3809,Y -133.0534,Z 184,A -76.527,B 3.7653,C 0.3372,E1 3.8067,E2 529.2525} C_DIS
LIN {X 16.898,Y -133.5417,Z 184,A -78.067,B 3.7651,C 0.3384,E1 3.8024,E2 530.7989} C_DIS
LIN {X 12.2299,Y -134.0496,Z 184,A -80.3067,B 3.7648,C 0.3414,E1 3.7961,E2 533.0705} C_DIS
LIN {X 8.8949,Y -134.3125,Z 184,A -81.3351,B 3.7651,C 0.3384,E1 3.7933,E2 534.049} C_DIS
LIN {X 5.3953,Y -134.4973,Z 184,A -82.961,B 3.765,C 0.34,E1 3.7887,E2 535.6929} C_DIS
LIN {X 0.9672,Y -134.6001,Z 184,A -84.872,B 3.765,C 0.3406,E1 3.7834,E2 537.6079} C_DIS
Enddeposition()
LIN {X 0.9672,Y -134.6001,Z 184,A -84.872,B 3.765,C 0.3406,E1 3.7834,E2 537.6079} C_DIS
Startdeposition()
$VEL.CP = VEL_PRINT
LIN {X 1.5665,Y -135.4989,Z 184,A -83.7733,B 3.7654,C 0.3353,E1 3.7867,E2 536.4309} C_DIS
LIN {X 4.7962,Y -135.4222,Z 184,A -82.1918,B 3.7656,C 0.333,E1 3.7911,E2 534.8204} C_DIS
LIN {X 8.1443,Y -135.2613,Z 184,A -80.9611,B 3.7654,C 0.3342,E1 3.7945,E2 533.6135} C_DIS
LIN {X 15.0125,Y -134.6729,Z 184,A -78.1932,B 3.7654,C 0.3344,E1 3.8022,E2 530.8634} C_DIS
LIN {X 18.8699,Y -134.1861,Z 184,A -76.5139,B 3.7655,C 0.3332,E1 3.8068,E2 529.1786} C_DIS
LIN {X 21.8206,Y -133.7384,Z 184,A -74.9059,B 3.7659,C 0.3292,E1 3.8114,E2 527.5243} C_DIS
LIN {X 25.6176,Y -133.0625,Z 184,A -73.6742,B 3.7657,C 0.3319,E1 3.8146,E2 526.3441} C_DIS
LIN {X 29.7478,Y -132.201,Z 184,A -71.9384,B 3.7657,C 0.331,E1 3.8194,E2 524.6136} C_DIS
LIN {X 33.0346,Y -131.4179,Z 184,A -70.5359,B 3.7658,C 0.3301,E1 3.8232,E2 523.2136} C_DIS
LIN {X 36.1986,Y -130.5817,Z 184,A -69.1661,B 3.7659,C 0.329,E1 3.8268,E2 521.8448} C_DIS
LIN {X 39.8491,Y -129.5142,Z 184,A -67.5398,B 3.7661,C 0.3273,E1 3.8312,E2 520.215} C_DIS
LIN {X 43.3576,Y -128.3833,Z 184,A -65.9658,B 3.7662,C 0.3256,E1 3.8354,E2 518.638} C_DIS
LIN {X 46.7205,Y -127.1993,Z 184,A -64.4243,B 3.7664,C 0.3236,E1 3.8395,E2 517.091} C_DIS
LIN {X 50.5207,Y -125.7357,Z 184,A -62.8594,B 3.7664,C 0.3232,E1 3.8435,E2 515.5454} C_DIS
LIN {X 53.432,Y -124.5269,Z 184,A -61.4823,B 3.7666,C 0.3211,E1 3.847,E2 514.1616} C_DIS
LIN {X 56.664,Y -123.0895,Z 184,A -60.1131,B 3.7666,C 0.3204,E1 3.8505,E2 512.8078} C_DIS
LIN {X 59.5652,Y -121.7125,Z 184,A -58.8851,B 3.7666,C 0.3199,E1 3.8535,E2 511.5959} C_DIS
LIN {X 62.1849,Y -120.397,Z 184,A -57.3663,B 3.7671,C 0.3153,E1 3.8574,E2 510.0398} C_DIS
LIN {X 65.3638,Y -118.7013,Z 184,A -55.9895,B 3.7671,C 0.3146,E1 3.8607,E2 508.681} C_DIS
LIN {X 70.7086,Y -115.597,Z 184,A -53.4317,B 3.7674,C 0.3111,E1 3.8669,E2 506.1286} C_DIS
LIN {X 74.142,Y -113.4258,Z 184,A -51.683,B 3.7677,C 0.308,E1 3.871,E2 504.3744} C_DIS
LIN {X 77.714,Y -111.0091,Z 184,A -50.1122,B 3.7677,C 0.3075,E1 3.8746,E2 502.8352} C_DIS
LIN {X 81.855,Y -107.9915,Z 184,A -47.7809,B 3.7682,C 0.302,E1 3.8799,E2 500.4807} C_DIS
LIN {X 84.579,Y -105.8715,Z 184,A -46.1205,B 3.7686,C 0.2971,E1 3.8835,E2 498.7929} C_DIS
LIN {X 87.3174,Y -103.6247,Z 184,A -44.9008,B 3.7686,C 0.2972,E1 3.8861,E2 497.6084} C_DIS
LIN {X 90.3496,Y -100.9915,Z 184,A -42.9512,B 3.769,C 0.2912,E1 3.8902,E2 495.6246} C_DIS
LIN {X 93.1851,Y -98.3815,Z 184,A -41.7398,B 3.769,C 0.2924,E1 3.8926,E2 494.4664} C_DIS
LIN {X 97.6377,Y -93.9647,Z 184,A -39.0533,B 3.7694,C 0.2865,E1 3.8979,E2 491.7733} C_DIS
LIN {X 100.0219,Y -91.4226,Z 184,A -37.4662,B 3.7697,C 0.2821,E1 3.9009,E2 490.1702} C_DIS
Enddeposition()
END
